// TIA Portal project "Polinka_3P_kwalifikacje_V16" (V16)

(* hardware
DEVICE "S7-1200 station_1"  S7-1200 Station
   slot 0: "Rack_0"  S7-1200 Rack  Rack  V1.0
   slot 1: "Polinka_Model"  CPU 1215C DC/DC/DC  6ES7 215-1AG40-0XB0  V4.2
DEVICE "S7-1200 station_2"  S7-1200 Station
   slot 0: "Rack_0"  S7-1200 Rack  Rack  V1.0
   slot 1: "Sterownik_do_zaprogramowania"  CPU 1215C DC/DC/DC  6ES7 215-1AG40-0XB0  V4.2
DEVICE "Polinka_HMI"  KTP700 Basic PN
   slot 0: "Polinka_HMI"  KTP700 Basic PN  6AV2 123-2GB03-0AX0  15.0.0.0
   slot 1: "HMI_RT_1"  KTP700 Basic PN  6AV2 123-2GB03-0AX0  15.0.0.0
   slot 5: "Polinka_HMI.IE_CP_1"  PROFINET Interface  15.0.0.0
      slot 1: "PROFINET Interface_1"  PROFINET Interface
         slot 1: "Port_1"  Port
*)

// ===== PLC "Polinka_Model"  CPU 1215C DC/DC/DC =====

VAR_GLOBAL   // PLC tag table "Default tag table"
   "System_Byte" AT %MB1 : Byte;
   "FirstScan" AT %M1.0 : Bool;
   "DiagStatusUpdate" AT %M1.1 : Bool;
   "AlwaysTRUE" AT %M1.2 : Bool;
   "AlwaysFALSE" AT %M1.3 : Bool;
   "Clock_Byte" AT %MB0 : Byte;
   "Clock_10Hz" AT %M0.0 : Bool;
   "Clock_5Hz" AT %M0.1 : Bool;
   "Clock_2.5Hz" AT %M0.2 : Bool;
   "Clock_2Hz" AT %M0.3 : Bool;
   "Clock_1.25Hz" AT %M0.4 : Bool;
   "Clock_1Hz" AT %M0.5 : Bool;
   "Clock_0.625Hz" AT %M0.6 : Bool;
   "Clock_0.5Hz" AT %M0.7 : Bool;
   "Tag_1" AT %M100.0 : Bool;
   "Tag_2" AT %M111.0 : Bool;
END_VAR

DATA_BLOCK "DB"   // DB1
{ S7_Optimized_Access := 'TRUE' }
VERSION : 0.1
   VAR
      w1_x : Int;
      w1_y : Int;
      w1_v : Real := 5.0;
      w1_drzwi_dx : Int := 0;
      w1_drzwiL_dx : Int;
      w1_drzwiP_dx : Int;
      w1_liczba_pasażerów : Int := 0;
      w1_drzwi_zamknięte : Bool;
      w1_drzwi_otwarte : Bool;
      zero : Int := 0;
      w2_y : Int := 0;
      w2_v : Int := 0;
      w2_drzwi_dx : Int := 0;
      w2_drzwiL_dx : Int := 0;
      w2_drzwiP_dx : Int := 0;
      w2_liczba_pasażerów : Int := 0;
      w2_drzwi_zamknięte : Bool := 0;
      w2_drzwi_otwarte : Bool := 0;
      w2_x : Int := 0;
      prędkość_wiatru : Real := 1.5;
      temperatura : Real := 20.0;
      czas_do_odjazdu : Int := 60;
      stacjaA_silnik_prędkość_zadana : Real := 0.0;
      stacjaA_silnik_prędkość_odczytana : Real := 0.0;
      stacjaA_silnik_przegrzanie : Bool;
      stacjaA_prędkość_odczytana : Real := 0.0;
      stacjaB_prędkość_odczytana : Real := 0.0;
      stacjaA_hamulec : Bool := false;
      stacjaB_hamulec : Bool := false;
      stacjaA_cz_A1 : Bool := false;
      stacjaA_cz_A2 : Bool := false;
      stacjaB_cz_B1 : Bool := false;
      stacjaB_cz_B2 : Bool := false;
      w1_d : Real := 0.0;
      w2_d : Real := 0.0;
      stacjaA_pasażer_0 : Bool := false;
      "stacjaA_pasażer+1" : Bool := false;
      "stacjaA_pasażer-1" : Bool := false;
      stacjaA_pasażerUP : Bool;
      stacjaA_pasażerDOWN : Bool;
      stacjaB_pasażer_0 : Bool := false;
      "stacjaB_pasażer+1" : Bool := false;
      "stacjaB_pasażer-1" : Bool := false;
      stacjaB_pasażerUP : Bool;
      stacjaB_pasażerDOWN : Bool;
      klawiatura : Word;
      awaria5 : Bool := false;
      awaria4 : Bool := false;
      awaria3 : Bool := false;
      awaria2 : Bool := false;
      awaria1 : Bool := false;
   END_VAR
BEGIN
END_DATA_BLOCK

DATA_BLOCK "Polinka_DB"   // DB2
{ S7_Optimized_Access := 'FALSE' }
VERSION : 0.1
   VAR
      st_stacjaA_silnik_prędkość : Real := 0.0;   // sterowanie prędkością silnika
      st_stacjaA_hamulec : Bool := true;   // sterowanie: 1 - hamulec włączony; 0 - wyłączony w stacji A
      st_stacjaA_zielone : Bool := false;   // sygnalizacja świetlna: 1-dozwolone wejście do wagonika
      st_stacjaA_czerwone : Bool := false;   // sygnalizacja świetlna: 1-zabronione wejście do wagonika
      st_stacjaB_hamulec : Bool := true;   // sterowanie: 1 - hamulec włączony; 0 - wyłączony w stacji B
      st_stacjaB_zielone : Bool := false;   // sygnalizacja świetlna: 1-dozwolone wejście do wagonika
      st_stacjaB_czerwone : Bool := false;   // sygnalizacja świetlna: 1-zabronione wejście do wagonika
      st_wagonik1_drzwi_zamykaj : Bool := false;   // 1 - zamykaj drzwi w wagoniku 1
      st_wagonik1_drzwi_otwieraj : Bool := false;   // 1 - otwieraj drzwi w wagoniku 1
      st_wagonik2_drzwi_zamykaj : Bool := false;   // 1 - zamykaj drzwi w wagoniku 2
      st_wagonik2_drzwi_otwieraj : Bool := false;   // 1 - otwieraj drzwi w wagoniku 2
      st_czas_do_odjazdu : Int := 60;   // czas pozostały do odjazdu wagoników
      st_kontrolka_STOP : Bool := false;   // 1 - podświetlaj przycisk "STOP"
      st_kontrolka_AUTO : Bool := false;   // 1 - podświetlaj przycisk "AUTO"
      st_kontrolka_RĘCZNIE : Bool := false;   // 1 - podświetlaj przycisk "RĘCZNIE"
      cz_wagonik1_położenie : Real;   // położenie wagonika 1, 0m - w stacji A, 756m - w stacji B
      "cz_wagonik1_l.pasażerów" : Int;   // liczba pasażerów w wagoniku 1
      cz_wagonik1_DZ : Bool;   // 1 gdy Drzwi w pełni Zamknięte i zabezpieczone
      cz_wagonik1_DO : Bool;   // 1 gdy Drzwi w pełni Otwarte i zabezpieczone
      cz_wagonik2_położenie : Real;   // położenie wagonika 2, 0m - w stacji A, 756m - w stacji B
      "cz_wagonik2_l.pasażerów" : Int;   // liczba pasażerów w wagoniku 2
      cz_wagonik2_DZ : Bool;   // 1 gdy Drzwi w pełni Zamknięte i zabezpieczone
      cz_wagonik2_DO : Bool;   // 1 gdy Drzwi w pełni Otwarte i zabezpieczone
      "cz_stacjaA_prędkość_(silnik)" : Real;   // prędkość liny napędowej odczytana na wale silnika [m/s]
      cz_stacjaA_prędkość : Real;   // prędkość liny napędowej odczytana w stacji A [m/s]
      cz_stacjaA_temperatura : Real;   // temperatura zewnętrzna
      cz_stacjaA_wiatr : Real;   // prędkość wiatru
      cz_stacjaA_silnik_przegrzanie : Bool;   // 1: działanie zabezpieczenia termicznego silnika
      cz_stacjaA_A1 : Bool;   // 1: wagonik na przystanku w stacji A
      cz_stacjaA_A2 : Bool;   // 1: wykolejona lina napędowa na słupie w stacji A
      cz_stacjaB_prędkość : Real;   // prędkość liny napędowej odczytana w stacji B [m/s]
      cz_stacjaB_B1 : Bool;   // 1: wagonik na przystanku w stacji B
      cz_stacjaB_B2 : Bool;   // 1: wykolejona lina napędowa na słupie w stacji B
      p_STOP : Bool;   // przycisk monostabilny STOP
      p_AUTO : Bool;   // przycisk monostabilny AUTO
      p_RĘCZNE : Bool;   // przycisk monostabilny RĘCZNIE
      "p_prędkość-20" : Bool;   // przycisk monostabilny -20 m/s
      "p_prędkość-5" : Bool;   // przycisk monostabilny -5 m/s
      p_prędkość_0 : Bool;   // przycisk monostabilny 0 m/s
      "p_prędkość+5" : Bool;   // przycisk monostabilny +5 m/s
      "p_prędkość+20" : Bool;   // przycisk monostabilny +20 m/s
      p_hamulecA_zał : Bool;   // przycisk monostabilny Hamulec A załącz
      p_hamulecA_wył : Bool;   // przycisk monostabilny Hamulec A wyłącz
      p_hamulecB_zał : Bool;   // przycisk monostabilny Hamulec B załącz
      p_hamulecB_wył : Bool;   // przycisk monostabilny Hamulec B wyłącz
      p_wagonik1_otw : Bool;   // przycisk mono.: otwieraj drzwi w wagoniku 1
      p_wagonik1_zam : Bool;   // przycisk mono.: zamykaj drzwi w wagoniku 1
      p_wagonik2_otw : Bool;   // przycisk mono.: otwieraj drzwi w wagoniku 2
      p_wagonik2_zam : Bool;   // przycisk mono.: zamykaj drzwi w wagoniku 2
   END_VAR
BEGIN
END_DATA_BLOCK

FUNCTION "fun3_Ruch_wagoników" : Void   // FC1, SCL
{ S7_Optimized_Access := 'TRUE' }
VERSION : 0.1
   VAR_TEMP
      d1 : Real;
      d2 : Real;
      d3 : Real;
      d4 : Real;
      d5 : Real;
      v_skala : Real;
      dk : Real;
      d : Real;
   END_VAR
   VAR CONSTANT
      "dT" : Real := 0.1;   // krok czasowy symulacji modelu [sek]
   END_VAR
BEGIN
   #v_skala := 1.0;

   #d1 := 20.0;
   #d2 := 158.0;
   #d3 := 400.0;
   #d4 := 158.0;
   #d5 := 20.0;

   #d := #d1 + #d2 + #d3 + #d4 + #d5 - (#d2 - 124.0) - (#d4 - 124.0);

   // 1. wagonik 1 - żółty:
   "DB".w1_d := "DB".w1_d + "DB".w1_v * #v_skala * #dT;
   IF "DB".w1_d < -18 THEN
       "DB".w1_d := -18;
   END_IF;

   IF "DB".w1_d > #d1 + #d2 + #d3 + #d4 + #d5 + 18.0 THEN
       "DB".w1_d := #d1 + #d2 + #d3 + #d4 + #d5 + 18.0;
   END_IF;

   // ruch na stacji A
   IF "DB".w1_d < #d1 THEN
       "DB".w1_x := "DB".w1_d;
       "DB".w1_y := 0.0;
   END_IF;

   // od stacji A do lewego słupa
   IF ("DB".w1_d >= #d1) AND ("DB".w1_d < #d1 + #d2)THEN
       #dk := "DB".w1_d - #d1;
       "DB".w1_y := -100.0 * #dk / #d2;
       "DB".w1_x := #d1 + 124.0 * #dk / #d2;
   END_IF;

   // między słupami
   IF ("DB".w1_d >= #d1 + #d2) AND ("DB".w1_d < #d1 + #d2 + #d3) THEN
       "DB".w1_x := "DB".w1_d - (#d2 - 124.0);
       "DB".w1_y := -100.0;
   END_IF;

   // od prawego słupa do stacji B
   IF ("DB".w1_d >= #d1 + #d2 + #d3) AND ("DB".w1_d < #d1 + #d2 + #d3 + #d4) THEN
       #dk := "DB".w1_d - #d1 - #d2 - #d3;
       "DB".w1_y := -100.0 + 100.0 * #dk / #d4;

       "DB".w1_x := "DB".w1_d - (#d2 - 124.0) + 124.0 * #dk / #d4;
       "DB".w1_x := #d1 + (#d2 - 34.0) + #d3 + 124.0 * #dk / #d4;
   END_IF;

   // ruch na stacji B
   IF ("DB".w1_d >= #d1 + #d2 + #d3 + #d4) THEN
       "DB".w1_x := "DB".w1_d - (#d2 - 124.0) - (#d4 - 124.0);
       "DB".w1_y := 0.0;
   END_IF;


   //  wagonik 2 - czerwony:
   "DB".w2_y := "DB".w1_y;
   "DB".w2_x := #d - "DB".w1_x;
   "DB".w2_x := -"DB".w1_x;
   "DB".w2_d := #d1 + #d2 + #d3 + #d4 + #d5 - "DB".w1_d;


   //krańcówki cz_A1 i cz_A2
   IF ("DB".w1_d <= 0) OR ("DB".w2_d <= 0) THEN
       "DB".stacjaA_cz_A1 := TRUE;
   ELSE
       "DB".stacjaA_cz_A1 := FALSE;
   END_IF;

   IF ("DB".w1_d >= 756) OR ("DB".w2_d >= 756) THEN
       "DB".stacjaB_cz_B1 := TRUE;
   ELSE
       "DB".stacjaB_cz_B1 := FALSE;
   END_IF;
END_FUNCTION

FUNCTION "fun4_Drzwi_wagoników" : Void   // FC2, SCL
{ S7_Optimized_Access := 'TRUE' }
VERSION : 0.1
BEGIN
   // wagonik 1 - drzwi:
   IF "Polinka_DB".st_wagonik1_drzwi_otwieraj THEN
       "DB".w1_drzwi_dx := "DB".w1_drzwi_dx + 1;
   END_IF;

   IF "Polinka_DB".st_wagonik1_drzwi_zamykaj THEN
       "DB".w1_drzwi_dx := "DB".w1_drzwi_dx - 1;
   END_IF;

   "DB".w1_drzwi_zamknięte := FALSE;
   "DB".w1_drzwi_otwarte := FALSE;
   IF "DB".w1_drzwi_dx <=0 THEN
       "DB".w1_drzwi_dx := 0;
       "DB".w1_drzwi_zamknięte := true;
   END_IF;

   IF "DB".w1_drzwi_dx >= 14 THEN
       "DB".w1_drzwi_dx := 14;
       "DB".w1_drzwi_otwarte := true;
   END_IF;

   "DB".w1_drzwiP_dx := "DB".w1_x + "DB".w1_drzwi_dx;
   "DB".w1_drzwiL_dx := "DB".w1_x - "DB".w1_drzwi_dx;

   // Błędne sterowanie (obie linie aktywne):
   IF "Polinka_DB".st_wagonik1_drzwi_zamykaj AND "Polinka_DB".st_wagonik1_drzwi_otwieraj THEN
       "DB".w1_drzwi_zamknięte := TRUE;
       "DB".w1_drzwi_otwarte := TRUE;
   END_IF;



   // wagonik 2 - drzwi:
   IF "Polinka_DB".st_wagonik2_drzwi_otwieraj THEN
       "DB".w2_drzwi_dx := "DB".w2_drzwi_dx + 1;
   END_IF;

   IF "Polinka_DB".st_wagonik2_drzwi_zamykaj THEN
       "DB".w2_drzwi_dx := "DB".w2_drzwi_dx - 1;
   END_IF;

   "DB".w2_drzwi_zamknięte := FALSE;
   "DB".w2_drzwi_otwarte := FALSE;
   IF "DB".w2_drzwi_dx <= 0 THEN
       "DB".w2_drzwi_dx := 0;
       "DB".w2_drzwi_zamknięte := true;
   END_IF;

   IF "DB".w2_drzwi_dx >= 14 THEN
       "DB".w2_drzwi_dx := 14;
       "DB".w2_drzwi_otwarte := true;
   END_IF;

   "DB".w2_drzwiP_dx := "DB".w2_x + "DB".w2_drzwi_dx;
   "DB".w2_drzwiL_dx := "DB".w2_x - "DB".w2_drzwi_dx;

   // Błędne sterowanie (obie linie aktywne):
   IF "Polinka_DB".st_wagonik2_drzwi_zamykaj AND "Polinka_DB".st_wagonik2_drzwi_otwieraj THEN
       "DB".w2_drzwi_zamknięte := TRUE;
       "DB".w2_drzwi_otwarte := TRUE;
   END_IF;



   ///
   (*
   // wagonik 1 - drzwi:
   IF "Polinka_DB".st_wagonik1_drzwi_otwieraj THEN
       "DB".w1_drzwi_dx := "DB".w1_drzwi_dx + 1;
   END_IF;

   IF "Polinka_DB".st_wagonik1_drzwi_zamykaj THEN
       "DB".w1_drzwi_dx := "DB".w1_drzwi_dx - 1;
   END_IF;

   "Polinka_DB".cz_wagonik1_DZ := FALSE;
   "Polinka_DB".cz_wagonik1_DO := FALSE;
   IF "DB".w1_drzwi_dx <=0 THEN
       "DB".w1_drzwi_dx := 0;
       "Polinka_DB".cz_wagonik1_DZ := true;
   END_IF;

   IF "DB".w1_drzwi_dx >= 14 THEN
       "DB".w1_drzwi_dx := 14;
       "Polinka_DB".cz_wagonik1_DO := true;
   END_IF;

   "DB".w1_drzwiP_dx := "DB".w1_x + "DB".w1_drzwi_dx;
   "DB".w1_drzwiL_dx := "DB".w1_x - "DB".w1_drzwi_dx;

   // Błędne sterowanie (obie linie aktywne):
   IF "Polinka_DB".st_wagonik1_drzwi_zamykaj AND "Polinka_DB".st_wagonik1_drzwi_otwieraj THEN
       "Polinka_DB".cz_wagonik1_DZ := TRUE;
       "Polinka_DB".cz_wagonik1_DO := TRUE;
   END_IF;



   // wagonik 2 - drzwi:
   IF "Polinka_DB".st_wagonik2_drzwi_otwieraj THEN
       "DB".w2_drzwi_dx := "DB".w2_drzwi_dx + 1;
   END_IF;

   IF "Polinka_DB".st_wagonik2_drzwi_zamykaj THEN
       "DB".w2_drzwi_dx := "DB".w2_drzwi_dx - 1;
   END_IF;

   "Polinka_DB".cz_wagonik2_DZ := FALSE;
   "Polinka_DB".cz_wagonik2_DO := FALSE;
   IF "DB".w2_drzwi_dx <= 0 THEN
       "DB".w2_drzwi_dx := 0;
       "Polinka_DB".cz_wagonik2_DZ := true;
   END_IF;

   IF "DB".w2_drzwi_dx >= 14 THEN
       "DB".w2_drzwi_dx := 14;
       "Polinka_DB".cz_wagonik2_DO := true;
   END_IF;

   "DB".w2_drzwiP_dx := "DB".w2_x + "DB".w2_drzwi_dx;
   "DB".w2_drzwiL_dx := "DB".w2_x - "DB".w2_drzwi_dx;

   // Błędne sterowanie (obie linie aktywne):
   IF "Polinka_DB".st_wagonik2_drzwi_zamykaj AND "Polinka_DB".st_wagonik2_drzwi_otwieraj THEN
       "Polinka_DB".cz_wagonik2_DZ := TRUE;
       "Polinka_DB".cz_wagonik2_DO := TRUE;
   END_IF;
   *)
END_FUNCTION

FUNCTION "fun5_Pasażerowie" : Void   // FC3, SCL
{ S7_Optimized_Access := 'TRUE' }
VERSION : 0.1
BEGIN
   "DB".stacjaA_pasażerDOWN := FALSE;
   "DB".stacjaA_pasażerUP :=FALSE;
   "DB".stacjaB_pasażerDOWN := FALSE;
   "DB".stacjaB_pasażerUP := FALSE;

   (*
   IF "DB"."stacjaB_pasażer+1" OR "DB"."stacjaB_pasażer-1" OR "DB".stacjaB_pasażer_0 THEN
       "DB".czas_do_odjazdu := "DB".czas_do_odjazdu + 1;
   END_IF;
   *)


   // 1. wagonik 1 na stacji A:
   IF "DB".w1_d <= 0 (*AND "DB".w1_d >=-5*) THEN
       IF "Polinka_DB".cz_wagonik1_DO THEN

           "DB".stacjaA_pasażerDOWN := true;

           IF "DB"."stacjaA_pasażer-1" THEN
               "DB"."stacjaA_pasażer-1" := 0;
               "DB".w1_liczba_pasażerów := "DB".w1_liczba_pasażerów - 1;
               IF "DB".w1_liczba_pasażerów < 0 THEN
                   "DB".w1_liczba_pasażerów := 0;
               END_IF;
           END_IF;

           IF "DB"."stacjaA_pasażer_0" THEN
               "DB"."stacjaA_pasażer_0" := 0;
               "DB".w1_liczba_pasażerów := 0;
           END_IF;


           IF "Polinka_DB".st_stacjaA_zielone AND NOT  "Polinka_DB".st_stacjaA_czerwone THEN
               "DB".stacjaA_pasażerUP := true;
               IF "DB"."stacjaA_pasażer+1" THEN
                   "DB"."stacjaA_pasażer+1" := 0;
                   "DB".w1_liczba_pasażerów := "DB".w1_liczba_pasażerów + 1;
               END_IF;
           END_IF;

       END_IF;
   END_IF;


   // 2. wagonik 1 na stacji B:
   IF (*"DB".w1_d <= 762 AND*) "DB".w1_d >= 756 THEN
       IF "Polinka_DB".cz_wagonik1_DO THEN

           "DB".stacjaB_pasażerDOWN := true;

           IF "DB"."stacjaB_pasażer-1" THEN
               "DB"."stacjaB_pasażer-1" := 0;
               "DB".w1_liczba_pasażerów := "DB".w1_liczba_pasażerów - 1;
               IF "DB".w1_liczba_pasażerów < 0 THEN
                   "DB".w1_liczba_pasażerów := 0;
               END_IF;
           END_IF;

           IF "DB"."stacjaB_pasażer_0" THEN
               "DB"."stacjaB_pasażer_0" := 0;
               "DB".w1_liczba_pasażerów := 0;
           END_IF;


           IF "Polinka_DB".st_stacjaB_zielone AND NOT "Polinka_DB".st_stacjaB_czerwone THEN
               "DB".stacjaB_pasażerUP := true;
               IF "DB"."stacjaB_pasażer+1" THEN
                   "DB"."stacjaB_pasażer+1" := 0;
                   "DB".w1_liczba_pasażerów := "DB".w1_liczba_pasażerów + 1;
               END_IF;
           END_IF;

       END_IF;
   END_IF;


   // 3. wagonik 2 na stacji A:
   IF "DB".w2_d <= 0 (*AND "DB".w2_d >= -5*) THEN
       IF "Polinka_DB".cz_wagonik2_DO THEN

           "DB".stacjaA_pasażerDOWN := true;

           IF "DB"."stacjaA_pasażer-1" THEN
               "DB"."stacjaA_pasażer-1" := 0;
               "DB".w2_liczba_pasażerów := "DB".w2_liczba_pasażerów - 1;
               IF "DB".w2_liczba_pasażerów < 0 THEN
                   "DB".w2_liczba_pasażerów := 0;
               END_IF;
           END_IF;

           IF "DB"."stacjaA_pasażer_0" THEN
               "DB"."stacjaA_pasażer_0" := 0;
               "DB".w2_liczba_pasażerów := 0;
           END_IF;


           IF "Polinka_DB".st_stacjaA_zielone AND NOT "Polinka_DB".st_stacjaA_czerwone THEN
               "DB".stacjaA_pasażerUP := true;
               IF "DB"."stacjaA_pasażer+1" THEN
                   "DB"."stacjaA_pasażer+1" := 0;
                   "DB".w2_liczba_pasażerów := "DB".w2_liczba_pasażerów + 1;
               END_IF;
           END_IF;

       END_IF;
   END_IF;


   // 4. wagonik 2 na stacji B:
   IF (*"DB".w2_d <= 762 AND*) "DB".w2_d >= 756 THEN
       IF "Polinka_DB".cz_wagonik2_DO THEN

           "DB".stacjaB_pasażerDOWN := true;

           IF "DB"."stacjaB_pasażer-1" THEN
               "DB"."stacjaB_pasażer-1" := 0;
               "DB".w2_liczba_pasażerów := "DB".w2_liczba_pasażerów - 1;
               IF "DB".w2_liczba_pasażerów < 0 THEN
                   "DB".w2_liczba_pasażerów := 0;
               END_IF;
           END_IF;

           IF "DB"."stacjaB_pasażer_0" THEN
               "DB"."stacjaB_pasażer_0" := 0;
               "DB".w2_liczba_pasażerów := 0;
           END_IF;


           IF "Polinka_DB".st_stacjaB_zielone AND NOT "Polinka_DB".st_stacjaB_czerwone THEN
               "DB".stacjaB_pasażerUP := true;
               IF "DB"."stacjaB_pasażer+1" THEN
                   "DB"."stacjaB_pasażer+1" := 0;
                   "DB".w2_liczba_pasażerów := "DB".w2_liczba_pasażerów + 1;
               END_IF;
           END_IF;

       END_IF;
   END_IF;



   (*        
   "DB"."stacjaA_pasażer+1" := 0;
   "DB"."stacjaA_pasażer-1" := 0;
   "DB"."stacjaA_pasażer_0" := 0;
   "DB"."stacjaB_pasażer+1" := 0;
   "DB"."stacjaB_pasażer-1" := 0;
   "DB"."stacjaB_pasażer_0" := 0;
   *)
END_FUNCTION

FUNCTION "fun6_SynchronizujDB_OUT" : Void   // FC4, SCL
{ S7_Optimized_Access := 'TRUE' }
VERSION : 0.1
   VAR_TEMP
      "a" : Word;
   END_VAR
BEGIN
   (*
   //1. synchronizacja z PLC_2 do modelu
   // 1.1 prędkości
   "DB".stacjaA_silnik_prędkość_zadana := "Polinka_DB".st_stacjaA_silnik_prędkość;
   "DB".stacjaA_silnik_prędkość_odczytana := "Polinka_DB".st_stacjaA_silnik_prędkość;
   "DB".stacjaA_prędkość_odczytana := "Polinka_DB".st_stacjaA_silnik_prędkość;
   "DB".stacjaB_prędkość_odczytana := "Polinka_DB".st_stacjaA_silnik_prędkość;

   // 1.2 hamulce
   "DB".stacjaA_hamulec := "Polinka_DB".st_stacjaA_hamulec;
   "DB".stacjaB_hamulec := "Polinka_DB".st_stacjaB_hamulec;

   // inne
   "DB".czas_do_odjazdu := "Polinka_DB".st_czas_do_odjazdu;
   *)


   /////////////////////////////////////////////////////////////////////////////////////
   //2. synchronizacja z modelu do PLC_2
   // 2.1 prędkości
   "Polinka_DB"."cz_stacjaA_prędkość_(silnik)" := "DB".stacjaA_silnik_prędkość_odczytana;
   "Polinka_DB"."cz_stacjaA_prędkość" := "DB".stacjaA_prędkość_odczytana;
   "Polinka_DB"."cz_stacjaB_prędkość" := "DB".stacjaB_prędkość_odczytana;


   // 2.2 informacje o wagonikach
   "Polinka_DB".cz_wagonik1_położenie := "DB".w1_d;
   "Polinka_DB".cz_wagonik2_położenie := "DB".w2_d;

   "Polinka_DB"."cz_wagonik1_l.pasażerów" := "DB".w1_liczba_pasażerów;
   "Polinka_DB"."cz_wagonik2_l.pasażerów" := "DB".w2_liczba_pasażerów;

   "Polinka_DB"."cz_wagonik1_DZ" := "DB".w1_drzwi_zamknięte;
   "Polinka_DB"."cz_wagonik1_DO" := "DB".w1_drzwi_otwarte;
   "Polinka_DB"."cz_wagonik2_DZ" := "DB".w2_drzwi_zamknięte;
   "Polinka_DB"."cz_wagonik2_DO" := "DB".w2_drzwi_otwarte;


   // 2.3 klawatura Panelu sterującego (do sterowania ręcznego)
   IF ("DB".klawiatura AND 1) > 0 THEN
       "Polinka_DB".p_STOP := 1;
   ELSE
       "Polinka_DB".p_STOP := 0;
   END_IF;

   IF ("DB".klawiatura AND 2) > 0 THEN
       "Polinka_DB".p_AUTO := 1;
   ELSE
       "Polinka_DB".p_AUTO := 0;
   END_IF;

   IF ("DB".klawiatura AND 4) > 0 THEN
       "Polinka_DB".p_RĘCZNE := 1;
   ELSE
       "Polinka_DB".p_RĘCZNE := 0;
   END_IF;

   IF ("DB".klawiatura AND 8) > 0 THEN
       "Polinka_DB"."p_prędkość-20" := 1;
   ELSE
       "Polinka_DB"."p_prędkość-20" := 0;
   END_IF;

   IF ("DB".klawiatura AND 16) > 0 THEN
       "Polinka_DB"."p_prędkość-5" := 1;
   ELSE
       "Polinka_DB"."p_prędkość-5" := 0;
   END_IF;

   IF ("DB".klawiatura AND 32) > 0 THEN
       "Polinka_DB"."p_prędkość_0" := 1;
   ELSE
       "Polinka_DB"."p_prędkość_0" := 0;
   END_IF;

   IF ("DB".klawiatura AND 64) > 0 THEN
       "Polinka_DB"."p_prędkość+5" := 1;
   ELSE
       "Polinka_DB"."p_prędkość+5" := 0;
   END_IF;

   IF ("DB".klawiatura AND 128) > 0 THEN
       "Polinka_DB"."p_prędkość+20" := 1;
   ELSE
       "Polinka_DB"."p_prędkość+20" := 0;
   END_IF;

   IF ("DB".klawiatura AND 256) > 0 THEN
       "Polinka_DB".p_hamulecA_zał := 1;
   ELSE
       "Polinka_DB".p_hamulecA_zał := 0;
   END_IF;

   IF ("DB".klawiatura AND 512) > 0 THEN
       "Polinka_DB".p_hamulecA_wył := 1;
   ELSE
       "Polinka_DB".p_hamulecA_wył := 0;
   END_IF;

   IF ("DB".klawiatura AND 1024) > 0 THEN
       "Polinka_DB".p_hamulecB_zał := 1;
   ELSE
       "Polinka_DB".p_hamulecB_zał := 0;
   END_IF;

   IF ("DB".klawiatura AND 2048) > 0 THEN
       "Polinka_DB".p_hamulecB_wył := 1;
   ELSE
       "Polinka_DB".p_hamulecB_wył := 0;
   END_IF;

   IF ("DB".klawiatura AND 4096) > 0 THEN
       "Polinka_DB".p_wagonik1_otw := 1;
   ELSE
       "Polinka_DB".p_wagonik1_otw := 0;
   END_IF;

   IF ("DB".klawiatura AND 8192) > 0 THEN
       "Polinka_DB".p_wagonik1_zam := 1;
   ELSE
       "Polinka_DB".p_wagonik1_zam := 0;
   END_IF;

   IF ("DB".klawiatura AND 16384) > 0 THEN
       "Polinka_DB".p_wagonik2_otw := 1;
   ELSE
       "Polinka_DB".p_wagonik2_otw := 0;
   END_IF;

   IF ("DB".klawiatura AND 32768) > 0 THEN
       "Polinka_DB".p_wagonik2_zam := 1;
   ELSE
       "Polinka_DB".p_wagonik2_zam := 0;
   END_IF;




   // 2.4 inne
   "Polinka_DB".cz_stacjaA_temperatura := "DB".temperatura ;
   IF "DB".prędkość_wiatru < 0 THEN
       "DB".prędkość_wiatru := 0.0;
   END_IF;
   "Polinka_DB".cz_stacjaA_wiatr := "DB".prędkość_wiatru;
   "Polinka_DB".cz_stacjaA_silnik_przegrzanie := "DB".stacjaA_silnik_przegrzanie;

   "Polinka_DB".cz_stacjaA_A1 := "DB".stacjaA_cz_A1;
   "Polinka_DB".cz_stacjaA_A2 := "DB".stacjaA_cz_A2;
   "Polinka_DB".cz_stacjaB_B1 := "DB".stacjaB_cz_B1;
   "Polinka_DB".cz_stacjaB_B2 := "DB".stacjaB_cz_B2;
END_FUNCTION

FUNCTION "fun1_SynchronizujDB_IN" : Void   // FC5, SCL
{ S7_Optimized_Access := 'TRUE' }
VERSION : 0.1
BEGIN
   /////////////////////////////////////////////////////////////////////////////////////
   //1. synchronizacja DB z PLC_2 do modelu
   // 1.1 prędkości
   "DB".stacjaA_silnik_prędkość_zadana := "Polinka_DB".st_stacjaA_silnik_prędkość;
   "DB".stacjaA_silnik_prędkość_odczytana := "Polinka_DB".st_stacjaA_silnik_prędkość;
   "DB".stacjaA_prędkość_odczytana := "Polinka_DB".st_stacjaA_silnik_prędkość;
   "DB".stacjaB_prędkość_odczytana := "Polinka_DB".st_stacjaA_silnik_prędkość;
   "DB".w1_v := "DB".stacjaA_silnik_prędkość_odczytana;

   // 1.2 hamulce
   "DB".stacjaA_hamulec := "Polinka_DB".st_stacjaA_hamulec;
   "DB".stacjaB_hamulec := "Polinka_DB".st_stacjaB_hamulec;

   // inne
   "DB".czas_do_odjazdu := "Polinka_DB".st_czas_do_odjazdu;
END_FUNCTION

FUNCTION "fun2_Awarie" : Void   // FC6, SCL
{ S7_Optimized_Access := 'TRUE' }
VERSION : 0.1
BEGIN
   // Awaria 1. - wykolejenie liny na słupie przy stacji A
   IF "DB".awaria1 THEN
       "DB".stacjaA_cz_A2 := TRUE;
   ELSE
       "DB".stacjaA_cz_A2 := FALSE;
   END_IF;


   // Awaria 2. - przegrzany silnik
   IF "DB".awaria2 THEN
       "DB".stacjaA_silnik_przegrzanie := TRUE;
   ELSE
       "DB".stacjaA_silnik_przegrzanie := FALSE;
   END_IF;


   // Awaria 3. - uszkodzona prądniczka tachometryczna w stacji B
   IF "DB".awaria3 THEN
       "DB".stacjaB_prędkość_odczytana := 0;
   END_IF;


   // Awaria 4. - uszkodzona sprzęgło przy silniku (połowa prędkości zadanej na kołach napędowych)
   IF "DB".awaria4 THEN
       "DB".stacjaA_prędkość_odczytana := "DB".stacjaA_silnik_prędkość_odczytana / 3;
       "DB".stacjaB_prędkość_odczytana := "DB".stacjaA_silnik_prędkość_odczytana / 3;
       "DB".w1_v := "DB".stacjaA_silnik_prędkość_odczytana / 3;
   END_IF;


   // Awaria 5. - (brak)
END_FUNCTION

ORGANIZATION_BLOCK "Main"   // OB1, LAD, ProgramCycle
TITLE = "Main Program Sweep (Cycle)"
{ S7_Optimized_Access := 'TRUE' }
VERSION : 0.1
   VAR_INPUT
      Initial_Call : Bool;   // Initial call of this OB
      Remanence : Bool;   // =True, if remanent data are available
   END_VAR
BEGIN
END_ORGANIZATION_BLOCK

ORGANIZATION_BLOCK "Polinka_model_Cyclic"   // OB30, SCL, CyclicInterrupt
{ S7_Optimized_Access := 'TRUE' }
VERSION : 0.1
   VAR_INPUT
      Initial_Call : Bool;   // Initial call of this OB
      Event_Count : Int;   // Events discarded
   END_VAR
BEGIN

   "fun1_SynchronizujDB_IN"();

   "fun2_Awarie"();

   "fun3_Ruch_wagoników"();

   "fun4_Drzwi_wagoników"();

   "fun5_Pasażerowie"();

   "fun6_SynchronizujDB_OUT"();
END_ORGANIZATION_BLOCK

// ===== PLC "Sterownik_do_zaprogramowania"  CPU 1215C DC/DC/DC =====

VAR_GLOBAL   // PLC tag table "Default tag table"
   "Tag_1" AT %M1.0 : Bool;
   "Clock_Byte" AT %MB0 : Byte;
   "Clock_10Hz" AT %M0.0 : Bool;
   "Clock_5Hz" AT %M0.1 : Bool;
   "Clock_2.5Hz" AT %M0.2 : Bool;
   "Clock_2Hz" AT %M0.3 : Bool;
   "Clock_1.25Hz" AT %M0.4 : Bool;
   "Clock_1Hz" AT %M0.5 : Bool;
   "Clock_0.625Hz" AT %M0.6 : Bool;
   "Clock_0.5Hz" AT %M0.7 : Bool;
   "Mem_Clock_1Hz" AT %M1.5 : Bool;
   "get_done" AT %M10.0 : Bool;
   "send" AT %M10.1 : Bool;
   "put_done" AT %M10.2 : Bool;
   "mem_get_done" AT %M10.3 : Bool;
   "mem_put_done" AT %M10.4 : Bool;
END_VAR

DATA_BLOCK "Polinka_DB"   // DB2
{ S7_Optimized_Access := 'FALSE' }
VERSION : 0.1
   VAR
      st_stacjaA_silnik_prędkość : Real := 0.0;   // sterowanie prędkością silnika
      st_stacjaA_hamulec : Bool := true;   // sterowanie: 1 - hamulec włączony; 0 - wyłączony w stacji A
      st_stacjaA_zielone : Bool := false;   // sygnalizacja świetlna: 1-dozwolone wejście do wagonika
      st_stacjaA_czerwone : Bool := false;   // sygnalizacja świetlna: 1-zabronione wejście do wagonika
      st_stacjaB_hamulec : Bool := true;   // sterowanie: 1 - hamulec włączony; 0 - wyłączony w stacji B
      st_stacjaB_zielone : Bool := false;   // sygnalizacja świetlna: 1-dozwolone wejście do wagonika
      st_stacjaB_czerwone : Bool := false;   // sygnalizacja świetlna: 1-zabronione wejście do wagonika
      st_wagonik1_drzwi_zamykaj : Bool := false;   // 1 - zamykaj drzwi w wagoniku 1
      st_wagonik1_drzwi_otwieraj : Bool := false;   // 1 - otwieraj drzwi w wagoniku 1
      st_wagonik2_drzwi_zamykaj : Bool := false;   // 1 - zamykaj drzwi w wagoniku 2
      st_wagonik2_drzwi_otwieraj : Bool := false;   // 1 - otwieraj drzwi w wagoniku 2
      st_czas_do_odjazdu : Int := 60;   // czas pozostały do odjazdu wagoników
      st_kontrolka_STOP : Bool := false;   // 1 - podświetlaj przycisk "STOP"
      st_kontrolka_AUTO : Bool := true;   // 1 - podświetlaj przycisk "AUTO"
      st_kontrolka_RĘCZNIE : Bool := false;   // 1 - podświetlaj przycisk "RĘCZNIE"
      cz_wagonik1_położenie : Real;   // położenie wagonika 1, 0m - w stacji A, 756m - w stacji B
      "cz_wagonik1_l.pasażerów" : Int;   // liczba pasażerów w wagoniku 1
      cz_wagonik1_DZ : Bool;   // 1 gdy Drzwi w pełni Zamknięte i zabezpieczone
      cz_wagonik1_DO : Bool;   // 1 gdy Drzwi w pełni Otwarte i zabezpieczone
      cz_wagonik2_położenie : Real;   // położenie wagonika 2, 0m - w stacji A, 756m - w stacji B
      "cz_wagonik2_l.pasażerów" : Int;   // liczba pasażerów w wagoniku 2
      cz_wagonik2_DZ : Bool;   // 1 gdy Drzwi w pełni Zamknięte i zabezpieczone
      cz_wagonik2_DO : Bool;   // 1 gdy Drzwi w pełni Otwarte i zabezpieczone
      "cz_stacjaA_prędkość_(silnik)" : Real;   // prędkość liny napędowej odczytana na wale silnika [m/s]
      cz_stacjaA_prędkość : Real;   // prędkość liny napędowej odczytana w stacji A [m/s]
      cz_stacjaA_temperatura : Real;   // temperatura zewnętrzna
      cz_stacjaA_wiatr : Real;   // prędkość wiatru
      cz_stacjaA_silnik_przegrzanie : Bool;   // 1: działanie zabezpieczenia termicznego silnika
      cz_stacjaA_A1 : Bool;   // 1: wagonik na przystanku w stacji A
      cz_stacjaA_A2 : Bool;   // 1: wykolejona lina napędowa na słupie w stacji A
      cz_stacjaB_prędkość : Real;   // prędkość liny napędowej odczytana w stacji B [m/s]
      cz_stacjaB_B1 : Bool;   // 1: wagonik na przystanku w stacji B
      cz_stacjaB_B2 : Bool;   // 1: wykolejona lina napędowa na słupie w stacji B
      p_STOP : Bool;   // przycisk monostabilny STOP
      p_AUTO : Bool;   // przycisk monostabilny AUTO
      p_RĘCZNE : Bool;   // przycisk monostabilny RĘCZNIE
      "p_prędkość-20" : Bool;   // przycisk monostabilny -20 m/s
      "p_prędkość-5" : Bool;   // przycisk monostabilny -5 m/s
      p_prędkość_0 : Bool;   // przycisk monostabilny 0 m/s
      "p_prędkość+5" : Bool;   // przycisk monostabilny +5 m/s
      "p_prędkość+20" : Bool;   // przycisk monostabilny +20 m/s
      p_hamulecA_zał : Bool;   // przycisk monostabilny Hamulec A załącz
      p_hamulecA_wył : Bool;   // przycisk monostabilny Hamulec A wyłącz
      p_hamulecB_zał : Bool;   // przycisk monostabilny Hamulec B załącz
      p_hamulecB_wył : Bool;   // przycisk monostabilny Hamulec B wyłącz
      p_wagonik1_otw : Bool;   // przycisk mono.: otwieraj drzwi w wagoniku 1
      p_wagonik1_zam : Bool;   // przycisk mono.: zamykaj drzwi w wagoniku 1
      p_wagonik2_otw : Bool;   // przycisk mono.: otwieraj drzwi w wagoniku 2
      p_wagonik2_zam : Bool;   // przycisk mono.: zamykaj drzwi w wagoniku 2
   END_VAR
BEGIN
END_DATA_BLOCK

DATA_BLOCK "praca_automatyczna_DB"   // DB3
{ S7_Optimized_Access := 'TRUE' }
VERSION : 0.1
// stored: InstanceOfName praca_automatyczna
"praca_automatyczna"
BEGIN
END_DATA_BLOCK

DATA_BLOCK "zmienne_DB"   // DB5
{ S7_Optimized_Access := 'TRUE' }
VERSION : 0.1
   VAR
      kierunek_jazdy : SInt := 1;
      praca_auto : Bool := true;
      praca_reczna : Bool;
      STOP : Bool;
      "mem_p-5" : Bool;
      "mem_p-20" : Bool;
      "mem_p+5" : Bool;
      "mem_p+20" : Bool;
      unieruchomienie_wiatr : Bool;   // Jeżeli bit ma stan wysoki to kolejka zostaje unieruchomiona na jedenj ze stacji (monostabilny)
      predkosc_wagonika_mocny_wiatr : Real := 1.0;   // Prędkość wagonika, jeżeli mocno wieje. Ogranicznik 0.5
      unieruchomienie_temp : Bool;
      unieruchomienie : Bool;
      mem_p_STOP : Bool;
      mem_p_AUTO : Bool;
      uzyto_stop : Bool;
      AWARIA_1 : Bool;
      AWARIA_2 : Bool;
      AWARIA_3 : Bool;
      AWARIA_4 : Bool;
      blokada_AUTO : Bool;
      praca_reczna_ograniczona : Bool;
      do_stacji : Bool;
   END_VAR
BEGIN
END_DATA_BLOCK

DATA_BLOCK "obsluga_awarii_DB"   // DB6
{ S7_Optimized_Access := 'TRUE' }
VERSION : 0.1
// stored: InstanceOfName obsluga_awarii
"obsluga_awarii"
BEGIN
END_DATA_BLOCK

DATA_BLOCK "obsluga_awarii_polinka_DB"   // DB7
{ S7_Optimized_Access := 'TRUE' }
VERSION : 0.1
// stored: InstanceOfName obsluga_awarii_polinka
"obsluga_awarii_polinka"
BEGIN
END_DATA_BLOCK

FUNCTION_BLOCK "praca_automatyczna"   // FB1, LAD
{ S7_Optimized_Access := 'TRUE' }
VERSION : 0.1
   VAR
      czas_jazdy : Time;
      jazda : Bool;
      gotowi : Bool;
      IEC_Timer_0_Instance : TON_TIME;
      time_slow_down : Time;
      bylo_pelne : Bool;
   END_VAR
   VAR_TEMP   // added for the SCL form of the ladder/FBD networks
      _w1 : Bool;
   END_VAR
BEGIN

REGION Network 1
   // Odliczanie sekund, a gdy jedziemy mierzenie czasu
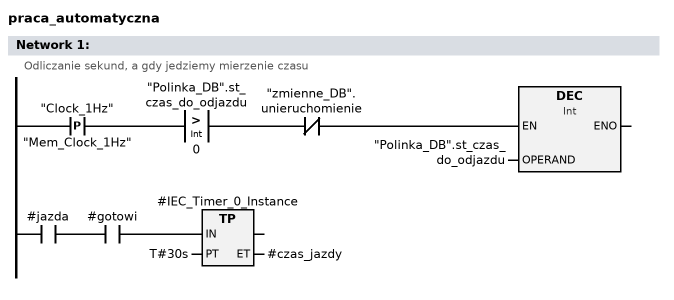
   #_w1 := "Clock_1Hz" AND NOT "Mem_Clock_1Hz";   // rising edge of "Clock_1Hz"
   "Mem_Clock_1Hz" := "Clock_1Hz";
   IF #_w1 AND ("Polinka_DB".st_czas_do_odjazdu > 0) AND NOT "zmienne_DB".unieruchomienie THEN
       "Polinka_DB".st_czas_do_odjazdu := "Polinka_DB".st_czas_do_odjazdu - 1;
   END_IF;
   #IEC_Timer_0_Instance(IN := #jazda AND #gotowi, PT := T#30s, ET => #czas_jazdy);   // TP
END_REGION

REGION Network 2 (SCL)
   // Jeśli skonczylo sie odliczanie, wagony nie są puste LUB jest 6 osób w obu wagonikach i nie #jazda to #jazda
   IF (("Polinka_DB".st_czas_do_odjazdu = 0 AND ("Polinka_DB"."cz_wagonik1_l.pasażerów" > 0 OR "Polinka_DB"."cz_wagonik2_l.pasażerów" > 0)) OR (("Polinka_DB"."cz_wagonik1_l.pasażerów" >= 6 AND "Polinka_DB"."cz_wagonik2_l.pasażerów" >= 6) AND NOT #bylo_pelne)) AND NOT #jazda AND NOT "zmienne_DB".unieruchomienie THEN
       #jazda := TRUE;
       "Polinka_DB".st_czas_do_odjazdu := 0;
       IF ("Polinka_DB"."cz_wagonik1_l.pasażerów" >= 6 AND "Polinka_DB"."cz_wagonik2_l.pasażerów" >= 6) THEN
           #bylo_pelne := TRUE;
       END_IF;
       // Zamknięcie drzwi w obu wagonikach
       "Polinka_DB".st_wagonik1_drzwi_otwieraj := 0;
       "Polinka_DB".st_wagonik2_drzwi_otwieraj := 0;
       "Polinka_DB".st_wagonik1_drzwi_zamykaj := 1;
       "Polinka_DB".st_wagonik2_drzwi_zamykaj := 1;
       // Zmiana światła na czerwone
       "Polinka_DB".st_stacjaA_zielone := 0;
       "Polinka_DB".st_stacjaA_czerwone := 1;
       "Polinka_DB".st_stacjaB_zielone := 0;
       "Polinka_DB".st_stacjaB_czerwone := 1;
       // Wyłączenie hamulcy
       "Polinka_DB".st_stacjaA_hamulec := 0;
       "Polinka_DB".st_stacjaB_hamulec := 0;
   // Gdy dalej trwa odliczanie:
   ELSIF NOT #jazda THEN
       // Drzwi otwarte w trakcie odliczania
       "Polinka_DB".st_wagonik1_drzwi_otwieraj := 1;
       "Polinka_DB".st_wagonik2_drzwi_otwieraj := 1;
       "Polinka_DB".st_wagonik1_drzwi_zamykaj := 0;
       "Polinka_DB".st_wagonik2_drzwi_zamykaj := 0;

       // Jeśli minął czas a nikogo nie ma to licz od początku
       IF "Polinka_DB".st_czas_do_odjazdu = 0 AND NOT ("Polinka_DB"."cz_wagonik1_l.pasażerów" > 0 OR "Polinka_DB"."cz_wagonik2_l.pasażerów" > 0) THEN
           "Polinka_DB".st_czas_do_odjazdu := 60;
       END_IF;
       // W zależności od kierunku jazdy wagoniki są na rożnych stacjach
       IF "zmienne_DB".kierunek_jazdy = 1 THEN
           // Jeśli pasażerów jest mniej niż 6 to zielone światło, w innym przypadku czerwone
           IF "Polinka_DB"."cz_wagonik1_l.pasażerów" < 6 THEN
               "Polinka_DB".st_stacjaA_zielone := 1;
               "Polinka_DB".st_stacjaA_czerwone := 0;
               #bylo_pelne := FALSE;
           ELSE
               "Polinka_DB".st_stacjaA_zielone := 0;
               "Polinka_DB".st_stacjaA_czerwone := 1;
           END_IF;
           IF "Polinka_DB"."cz_wagonik2_l.pasażerów" < 6 THEN
               "Polinka_DB".st_stacjaB_zielone := 1;
               "Polinka_DB".st_stacjaB_czerwone := 0;
               #bylo_pelne := FALSE;
           ELSE
               "Polinka_DB".st_stacjaB_zielone := 0;
               "Polinka_DB".st_stacjaB_czerwone := 1;
           END_IF;
       ELSE
           // Jeśli pasażerów jest mniej niż 6 to zielone światło, w innym przypadku czerwone
           IF "Polinka_DB"."cz_wagonik1_l.pasażerów" < 6 THEN
               "Polinka_DB".st_stacjaB_zielone := 1;
               "Polinka_DB".st_stacjaB_czerwone := 0;
               #bylo_pelne := FALSE;
           ELSE
               "Polinka_DB".st_stacjaB_zielone := 0;
               "Polinka_DB".st_stacjaB_czerwone := 1;
           END_IF;
           IF "Polinka_DB"."cz_wagonik2_l.pasażerów" < 6 THEN
               "Polinka_DB".st_stacjaA_zielone := 1;
               "Polinka_DB".st_stacjaA_czerwone := 0;
               #bylo_pelne := FALSE;
           ELSE
               "Polinka_DB".st_stacjaA_zielone := 0;
               "Polinka_DB".st_stacjaA_czerwone := 1;
           END_IF;
       END_IF;
   // Jeśli dojechał do końca to zatrzymaj, zmień kierunek oraz załącz hamulce
   ELSIF #jazda AND ("Polinka_DB".cz_stacjaA_A1 OR "Polinka_DB".cz_stacjaA_A2) AND #czas_jazdy > T#10s THEN
       #jazda := FALSE;
       "Polinka_DB".st_stacjaA_silnik_prędkość := 0;
       "zmienne_DB".kierunek_jazdy := - "zmienne_DB".kierunek_jazdy;
       "Polinka_DB".st_czas_do_odjazdu := 60;
       "Polinka_DB".st_czas_do_odjazdu := "Polinka_DB".st_czas_do_odjazdu + 1;
       // Załączenie hamulcy
       "Polinka_DB".st_stacjaA_hamulec := 1;
       "Polinka_DB".st_stacjaB_hamulec := 1;
   END_IF;
END_REGION

REGION Network 3 (SCL)
   // Gdy mamy jechać
   IF #jazda THEN
       // Najpierw sprawdzamy czy jesteśmy gotowi (zamknięte drzwi itp.)
       IF "Polinka_DB".cz_wagonik1_DZ AND "Polinka_DB".cz_wagonik2_DZ AND NOT "Polinka_DB".cz_wagonik1_DO
           AND NOT "Polinka_DB".cz_wagonik2_DO AND NOT "Polinka_DB".st_stacjaA_hamulec AND NOT "Polinka_DB".st_stacjaB_hamulec
           AND NOT "Polinka_DB".p_STOP THEN
           #gotowi := TRUE;
       ELSE
           #gotowi := FALSE;
       END_IF;
       // Gdy jesteśmy gotowi to w zależności od tego jak długo jedziemy tak zmieniamy prędkość
       IF #czas_jazdy < T#1s THEN
           #time_slow_down := T#0s;
           "Polinka_DB".st_stacjaA_silnik_prędkość := 0.0;
       ELSIF #czas_jazdy < T#2s THEN
           "Polinka_DB".st_stacjaA_silnik_prędkość := INT_TO_REAL("zmienne_DB".kierunek_jazdy) * 5.0;
       ELSIF #czas_jazdy < T#3s THEN
           "Polinka_DB".st_stacjaA_silnik_prędkość := INT_TO_REAL("zmienne_DB".kierunek_jazdy) * 25.0;
       ELSIF #czas_jazdy < T#4s THEN
           "Polinka_DB".st_stacjaA_silnik_prędkość := INT_TO_REAL("zmienne_DB".kierunek_jazdy) * 40.0;
       // Poniższy warunek oznacza tyle: wagonik jest dalej niż 70 m do celu
       ELSIF INT_TO_REAL("zmienne_DB".kierunek_jazdy) * "Polinka_DB".cz_wagonik1_położenie
           < INT_TO_REAL("zmienne_DB".kierunek_jazdy) * (378.0 + INT_TO_REAL("zmienne_DB".kierunek_jazdy) * 308.0) THEN
           "Polinka_DB".st_stacjaA_silnik_prędkość := INT_TO_REAL("zmienne_DB".kierunek_jazdy) * 50.0;
       // Odmierzamy czas od momentu gdy mamy zwalniać
       ELSIF #time_slow_down = T#0ms THEN
           #time_slow_down := #czas_jazdy;
       ELSIF #czas_jazdy < #time_slow_down + T#900ms THEN
           "Polinka_DB".st_stacjaA_silnik_prędkość := INT_TO_REAL("zmienne_DB".kierunek_jazdy) * 40.0;
       ELSIF #czas_jazdy < #time_slow_down + T#1900ms THEN
           "Polinka_DB".st_stacjaA_silnik_prędkość := INT_TO_REAL("zmienne_DB".kierunek_jazdy) * 25.0;
       ELSIF #czas_jazdy < #time_slow_down + T#2900ms THEN
           "Polinka_DB".st_stacjaA_silnik_prędkość := INT_TO_REAL("zmienne_DB".kierunek_jazdy) * 5.0;
       END_IF;
       "Polinka_DB".st_stacjaA_silnik_prędkość := "Polinka_DB".st_stacjaA_silnik_prędkość * "zmienne_DB".predkosc_wagonika_mocny_wiatr;
   END_IF;
END_REGION
END_FUNCTION_BLOCK

FUNCTION_BLOCK "Zadanie4"   // FB1, LAD
{ S7_Optimized_Access := 'TRUE' }
VERSION : 0.1
   VAR_INPUT
      cz_stacjaA_A2 : Bool;
      cz_stacjaA_silnik_przegrzanie : Bool;
      cz_stacjaA_prędkość : Real;
      cz_stacjaB_prędkość : Real;
      cz_stacjaA_A1 : Bool;
      cz_wagonik1_położenie : Real;
      pracaAuto : Bool;
      stacjaA_silnik_prędkość : Real;
      cz_stacjaA_prędkość_silnik : Real;
   END_VAR
   VAR_OUTPUT
      p_hamulecA_zal : Bool;
      p_hamulecA_Wyl : Bool;
      p_hamulecB_Wyl : Bool;
      p_hamulecB_zal : Bool;
      stopAwaryjny : Bool;
      blokadaPowrotuDoAuto : Bool;
      silnikPredkoscPrzeliczona : Real;
      reczneSterowanie : Bool;
   END_VAR
   VAR
      ALWAYS_ON : Bool := TRUE;
      setAwaria2 : Bool;
      setAwaria3 : Bool;
      manual1 : Bool;
      manual2 : Bool;
      resetAuto1 : Bool;
      resetAuto2 : Bool;
      speedADiv : Real;
      resetManual : Bool;
      speedBDiv : Real;
   END_VAR
   VAR_TEMP   // added for the SCL form of the ladder/FBD networks
      _w1 : Bool;
   END_VAR
BEGIN

REGION Network 1 (SCL): Przeliczenie wartości do porównania
   #speedADiv := #cz_stacjaA_prędkość_silnik / 3;
   #speedBDiv := #cz_stacjaA_prędkość_silnik / 3;
END_REGION

REGION Network 2: Załączenie blokady przejścia z trybu Manualnego do trybu automatyczneogo po Awarii
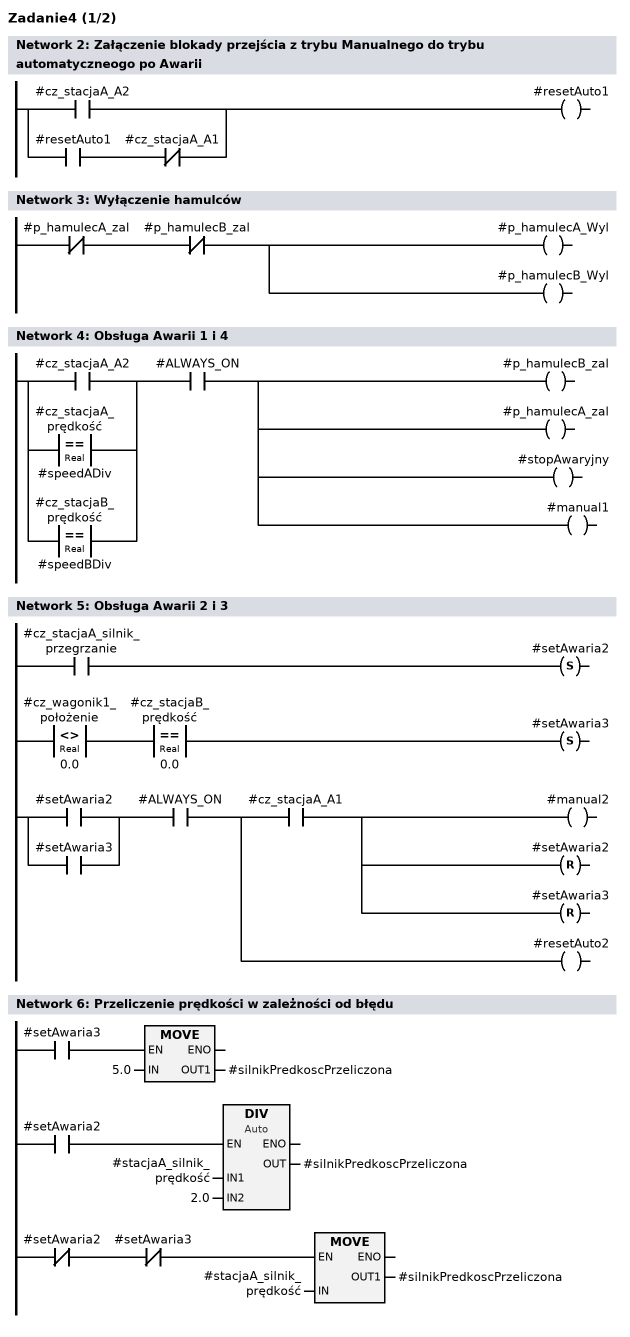
   RUNG wire#powerrail
      Contact( #cz_stacjaA_A2 )
      wire#w1
      Coil( #resetAuto1 )
   END_RUNG
   RUNG wire#powerrail
      Contact( #resetAuto1 )
      I_Contact( #cz_stacjaA_A1 )
   END_RUNG wire#w1
   // the same network as SCL:
   #resetAuto1 := #cz_stacjaA_A2 OR (#resetAuto1 AND NOT #cz_stacjaA_A1);
END_REGION

REGION Network 3: Wyłączenie hamulców
   RUNG wire#powerrail
      I_Contact( #p_hamulecA_zal )
      I_Contact( #p_hamulecB_zal )
      wire#w1
      Coil( #p_hamulecA_Wyl )
   END_RUNG
   RUNG wire#w1
      Coil( #p_hamulecB_Wyl )
   END_RUNG
   // the same network as SCL:
   #p_hamulecA_Wyl := NOT #p_hamulecA_zal AND NOT #p_hamulecB_zal;
   #p_hamulecB_Wyl := #p_hamulecA_Wyl;
END_REGION

REGION Network 4: Obsługa Awarii 1 i 4
   RUNG wire#powerrail
      Contact( #cz_stacjaA_A2 )
      wire#w1
      Contact( #ALWAYS_ON )
      wire#w2
      Coil( #p_hamulecB_zal )
   END_RUNG
   RUNG wire#powerrail
      { S7_Templates := "SrcType := Real" } EQ_Contact(in1 := #cz_stacjaA_prędkość, in2 := #speedADiv)
   END_RUNG wire#w1
   RUNG wire#powerrail
      { S7_Templates := "SrcType := Real" } EQ_Contact(in1 := #cz_stacjaB_prędkość, in2 := #speedBDiv)
   END_RUNG wire#w1
   RUNG wire#w2
      Coil( #p_hamulecA_zal )
   END_RUNG
   RUNG wire#w2
      Coil( #stopAwaryjny )
   END_RUNG
   RUNG wire#w2
      Coil( #manual1 )
   END_RUNG
   // the same network as SCL:
   #p_hamulecB_zal := (#cz_stacjaA_A2 OR (#cz_stacjaA_prędkość = #speedADiv) OR (#cz_stacjaB_prędkość = #speedBDiv)) AND #ALWAYS_ON;
   #p_hamulecA_zal := #p_hamulecB_zal;
   #stopAwaryjny := #p_hamulecB_zal;
   #manual1 := #p_hamulecB_zal;
END_REGION

REGION Network 5: Obsługa Awarii 2 i 3
   RUNG wire#powerrail
      Contact( #cz_stacjaA_silnik_przegrzanie )
      S_Coil( #setAwaria2 )
   END_RUNG
   RUNG wire#powerrail
      { S7_Templates := "SrcType := Real" } NE_Contact(in1 := #cz_wagonik1_położenie, in2 := 0.0)
      { S7_Templates := "SrcType := Real" } EQ_Contact(in1 := #cz_stacjaB_prędkość, in2 := 0.0)
      S_Coil( #setAwaria3 )
   END_RUNG
   RUNG wire#powerrail
      Contact( #setAwaria2 )
      wire#w1
      Contact( #ALWAYS_ON )
      wire#w2
      Contact( #cz_stacjaA_A1 )
      wire#w3
      Coil( #manual2 )
   END_RUNG
   RUNG wire#powerrail
      Contact( #setAwaria3 )
   END_RUNG wire#w1
   RUNG wire#w3
      R_Coil( #setAwaria2 )
   END_RUNG
   RUNG wire#w3
      R_Coil( #setAwaria3 )
   END_RUNG
   RUNG wire#w2
      Coil( #resetAuto2 )
   END_RUNG
   // the same network as SCL:
   IF #cz_stacjaA_silnik_przegrzanie THEN #setAwaria2 := TRUE; END_IF;
   IF (#cz_wagonik1_położenie <> 0.0) AND (#cz_stacjaB_prędkość = 0.0) THEN #setAwaria3 := TRUE; END_IF;
   #_w1 := (#setAwaria2 OR #setAwaria3) AND #ALWAYS_ON;
   #manual2 := #_w1 AND #cz_stacjaA_A1;
   IF #manual2 THEN
       #setAwaria2 := FALSE;
       #setAwaria3 := FALSE;
   END_IF;
   #resetAuto2 := #_w1;
END_REGION

REGION Network 6: Przeliczenie prędkości w zależności od błędu
   RUNG wire#powerrail
      Contact( #setAwaria3 )
      Move(in := 5.0, out1 => #silnikPredkoscPrzeliczona)
   END_RUNG
   RUNG wire#powerrail
      Contact( #setAwaria2 )
      Div(in1 := #stacjaA_silnik_prędkość, in2 := 2.0, out => #silnikPredkoscPrzeliczona)
   END_RUNG
   RUNG wire#powerrail
      I_Contact( #setAwaria2 )
      I_Contact( #setAwaria3 )
      Move(in := #stacjaA_silnik_prędkość, out1 => #silnikPredkoscPrzeliczona)
   END_RUNG
   // the same network as SCL:
   IF #setAwaria3 THEN #silnikPredkoscPrzeliczona := 5.0; END_IF;
   IF #setAwaria2 THEN #silnikPredkoscPrzeliczona := #stacjaA_silnik_prędkość / 2.0; END_IF;
   IF NOT #setAwaria2 AND NOT #setAwaria3 THEN
       #silnikPredkoscPrzeliczona := #stacjaA_silnik_prędkość;
   END_IF;
END_REGION

REGION Network 7: Zablokowanie przejścia z trybu Manualne do Automatycznego
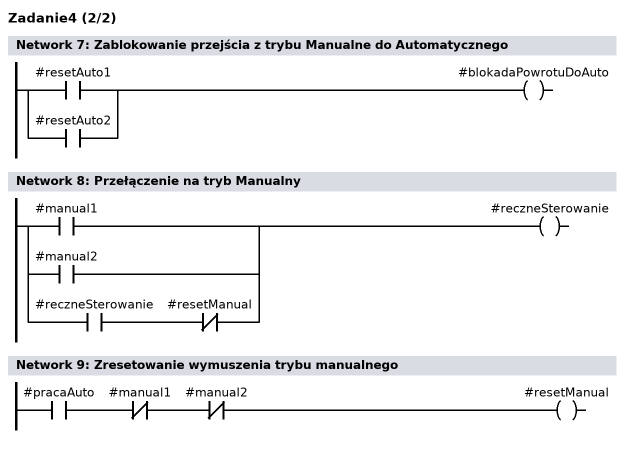
   RUNG wire#powerrail
      Contact( #resetAuto1 )
      wire#w1
      Coil( #blokadaPowrotuDoAuto )
   END_RUNG
   RUNG wire#powerrail
      Contact( #resetAuto2 )
   END_RUNG wire#w1
   // the same network as SCL:
   #blokadaPowrotuDoAuto := #resetAuto1 OR #resetAuto2;
END_REGION

REGION Network 8: Przełączenie na tryb Manualny
   RUNG wire#powerrail
      Contact( #manual1 )
      wire#w1
      Coil( #reczneSterowanie )
   END_RUNG
   RUNG wire#powerrail
      Contact( #manual2 )
   END_RUNG wire#w1
   RUNG wire#powerrail
      Contact( #reczneSterowanie )
      I_Contact( #resetManual )
   END_RUNG wire#w1
   // the same network as SCL:
   #reczneSterowanie := #manual1 OR #manual2 OR (#reczneSterowanie AND NOT #resetManual);
END_REGION

REGION Network 9: Zresetowanie wymuszenia trybu manualnego
   RUNG wire#powerrail
      Contact( #pracaAuto )
      I_Contact( #manual1 )
      I_Contact( #manual2 )
      Coil( #resetManual )
   END_RUNG
   // the same network as SCL:
   #resetManual := #pracaAuto AND NOT #manual1 AND NOT #manual2;
END_REGION
END_FUNCTION_BLOCK

FUNCTION_BLOCK "obsluga_awarii"   // FB2, LAD
{ S7_Optimized_Access := 'TRUE' }
VERSION : 0.1
   VAR_INPUT
      cz_stacjaA_A2 : Bool;
      cz_stacjaA_silnik_przegrzanie : Bool;
      cz_stacjaA_prędkość : Real;
      cz_stacjaB_prędkość : Real;
      cz_stacjaA_A1 : Bool;
      cz_wagonik1_położenie : Real;
      stacjaA_silnik_prędkość : Real;
      cz_stacjaA_prędkość_silnik : Real;
   END_VAR
   VAR_OUTPUT
      hamulecA_zal : Bool;
      hamulecB_zal : Bool;
      stopAwaryjny : Bool;
      blokadaPowrotuDoAuto : Bool;
      silnikPredkoscPrzeliczona : Real;
      reczneSterowanie : Bool;
      reczneOgraniczone : Bool;
   END_VAR
   VAR
      ALWAYS_ON : Bool := TRUE;
      setAwaria2 : Bool;
      setAwaria3 : Bool;
      manual1 : Bool;
      manual2 : Bool;
      resetAuto1 : Bool;
      resetAuto2 : Bool;
      speedADiv : Real;
      resetManual : Bool;
      speedBDiv : Real;
   END_VAR
BEGIN

REGION Network 1 (SCL): Przeliczenie wartości do porównania
   #speedADiv := #cz_stacjaA_prędkość_silnik / 3;
   #speedBDiv := #cz_stacjaA_prędkość_silnik / 3;
END_REGION

REGION Network 2: Załączenie blokady przejścia z trybu Manualnego do trybu automatyczneogo po Awarii
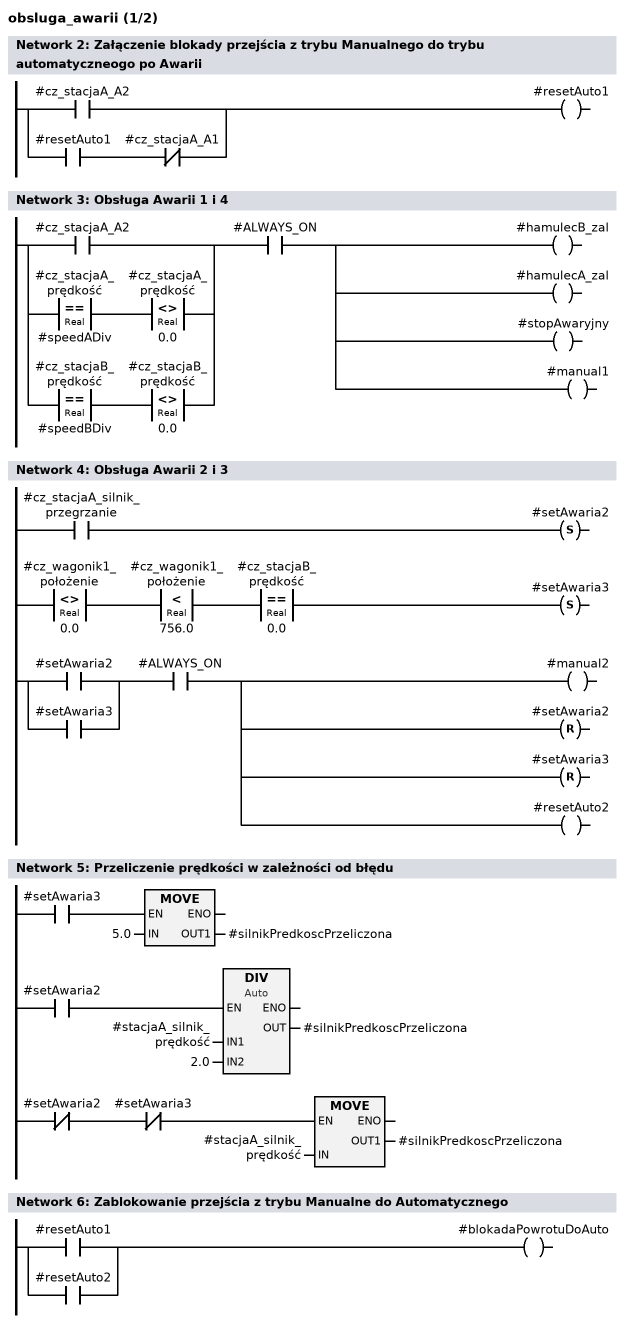
   RUNG wire#powerrail
      Contact( #cz_stacjaA_A2 )
      wire#w1
      Coil( #resetAuto1 )
   END_RUNG
   RUNG wire#powerrail
      Contact( #resetAuto1 )
      I_Contact( #cz_stacjaA_A1 )
   END_RUNG wire#w1
   // the same network as SCL:
   #resetAuto1 := #cz_stacjaA_A2 OR (#resetAuto1 AND NOT #cz_stacjaA_A1);
END_REGION

REGION Network 3: Obsługa Awarii 1 i 4
   RUNG wire#powerrail
      Contact( #cz_stacjaA_A2 )
      wire#w1
      Contact( #ALWAYS_ON )
      wire#w2
      Coil( #hamulecB_zal )
   END_RUNG
   RUNG wire#powerrail
      { S7_Templates := "SrcType := Real" } EQ_Contact(in1 := #cz_stacjaA_prędkość, in2 := #speedADiv)
      { S7_Templates := "SrcType := Real" } NE_Contact(in1 := #cz_stacjaA_prędkość, in2 := 0.0)
   END_RUNG wire#w1
   RUNG wire#powerrail
      { S7_Templates := "SrcType := Real" } EQ_Contact(in1 := #cz_stacjaB_prędkość, in2 := #speedBDiv)
      { S7_Templates := "SrcType := Real" } NE_Contact(in1 := #cz_stacjaB_prędkość, in2 := 0.0)
   END_RUNG wire#w1
   RUNG wire#w2
      Coil( #hamulecA_zal )
   END_RUNG
   RUNG wire#w2
      Coil( #stopAwaryjny )
   END_RUNG
   RUNG wire#w2
      Coil( #manual1 )
   END_RUNG
   // the same network as SCL:
   #hamulecB_zal := (#cz_stacjaA_A2 OR ((#cz_stacjaA_prędkość = #speedADiv) AND (#cz_stacjaA_prędkość <> 0.0)) OR ((#cz_stacjaB_prędkość = #speedBDiv) AND (#cz_stacjaB_prędkość <> 0.0))) AND #ALWAYS_ON;
   #hamulecA_zal := #hamulecB_zal;
   #stopAwaryjny := #hamulecB_zal;
   #manual1 := #hamulecB_zal;
END_REGION

REGION Network 4: Obsługa Awarii 2 i 3
   RUNG wire#powerrail
      Contact( #cz_stacjaA_silnik_przegrzanie )
      S_Coil( #setAwaria2 )
   END_RUNG
   RUNG wire#powerrail
      { S7_Templates := "SrcType := Real" } NE_Contact(in1 := #cz_wagonik1_położenie, in2 := 0.0)
      { S7_Templates := "SrcType := Real" } LT_Contact(in1 := #cz_wagonik1_położenie, in2 := 756.0)
      { S7_Templates := "SrcType := Real" } EQ_Contact(in1 := #cz_stacjaB_prędkość, in2 := 0.0)
      S_Coil( #setAwaria3 )
   END_RUNG
   RUNG wire#powerrail
      Contact( #setAwaria2 )
      wire#w1
      Contact( #ALWAYS_ON )
      wire#w2
      Coil( #manual2 )
   END_RUNG
   RUNG wire#powerrail
      Contact( #setAwaria3 )
   END_RUNG wire#w1
   RUNG wire#w2
      R_Coil( #setAwaria2 )
   END_RUNG
   RUNG wire#w2
      R_Coil( #setAwaria3 )
   END_RUNG
   RUNG wire#w2
      Coil( #resetAuto2 )
   END_RUNG
   // the same network as SCL:
   IF #cz_stacjaA_silnik_przegrzanie THEN #setAwaria2 := TRUE; END_IF;
   IF (#cz_wagonik1_położenie <> 0.0) AND (#cz_wagonik1_położenie < 756.0) AND (#cz_stacjaB_prędkość = 0.0) THEN
       #setAwaria3 := TRUE;
   END_IF;
   #manual2 := (#setAwaria2 OR #setAwaria3) AND #ALWAYS_ON;
   IF #manual2 THEN
       #setAwaria2 := FALSE;
       #setAwaria3 := FALSE;
   END_IF;
   #resetAuto2 := #manual2;
END_REGION

REGION Network 5: Przeliczenie prędkości w zależności od błędu
   RUNG wire#powerrail
      Contact( #setAwaria3 )
      Move(in := 5.0, out1 => #silnikPredkoscPrzeliczona)
   END_RUNG
   RUNG wire#powerrail
      Contact( #setAwaria2 )
      Div(in1 := #stacjaA_silnik_prędkość, in2 := 2.0, out => #silnikPredkoscPrzeliczona)
   END_RUNG
   RUNG wire#powerrail
      I_Contact( #setAwaria2 )
      I_Contact( #setAwaria3 )
      Move(in := #stacjaA_silnik_prędkość, out1 => #silnikPredkoscPrzeliczona)
   END_RUNG
   // the same network as SCL:
   IF #setAwaria3 THEN #silnikPredkoscPrzeliczona := 5.0; END_IF;
   IF #setAwaria2 THEN #silnikPredkoscPrzeliczona := #stacjaA_silnik_prędkość / 2.0; END_IF;
   IF NOT #setAwaria2 AND NOT #setAwaria3 THEN
       #silnikPredkoscPrzeliczona := #stacjaA_silnik_prędkość;
   END_IF;
END_REGION

REGION Network 6: Zablokowanie przejścia z trybu Manualne do Automatycznego
   RUNG wire#powerrail
      Contact( #resetAuto1 )
      wire#w1
      Coil( #blokadaPowrotuDoAuto )
   END_RUNG
   RUNG wire#powerrail
      Contact( #resetAuto2 )
   END_RUNG wire#w1
   // the same network as SCL:
   #blokadaPowrotuDoAuto := #resetAuto1 OR #resetAuto2;
END_REGION

REGION Network 7: Przełączenie na tryb Manualny
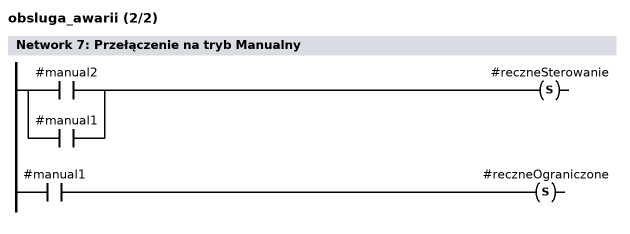
   RUNG wire#powerrail
      Contact( #manual2 )
      wire#w1
      S_Coil( #reczneSterowanie )
   END_RUNG
   RUNG wire#powerrail
      Contact( #manual1 )
   END_RUNG wire#w1
   RUNG wire#powerrail
      Contact( #manual1 )
      S_Coil( #reczneOgraniczone )
   END_RUNG
   // the same network as SCL:
   IF #manual2 OR #manual1 THEN #reczneSterowanie := TRUE; END_IF;
   IF #manual1 THEN #reczneOgraniczone := TRUE; END_IF;
END_REGION
END_FUNCTION_BLOCK

FUNCTION_BLOCK "obsluga_awarii_polinka"   // FB3, LAD
{ S7_Optimized_Access := 'TRUE' }
VERSION : 0.1
   VAR_TEMP   // added for the SCL form of the ladder/FBD networks
      _w1 : Bool;
   END_VAR
BEGIN

REGION Network 1
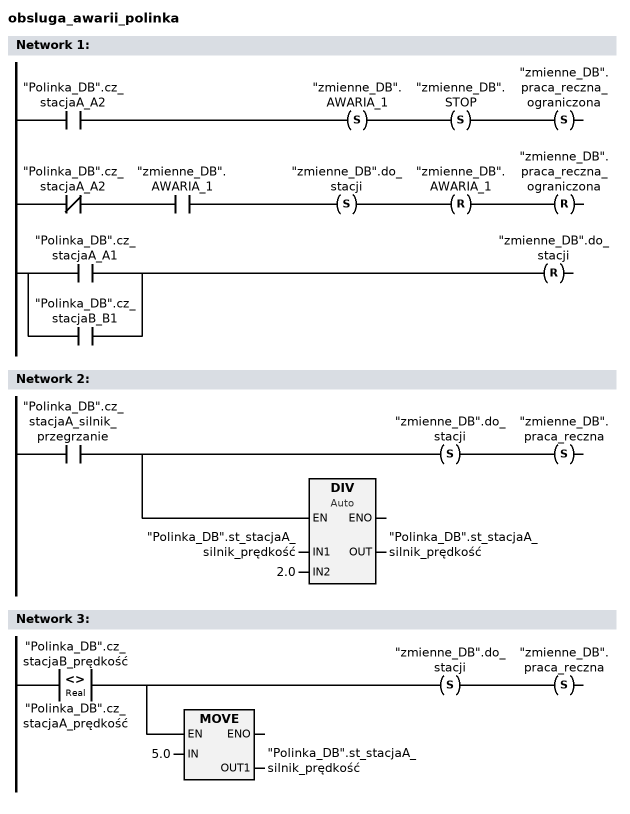
   RUNG wire#powerrail
      Contact( "Polinka_DB".cz_stacjaA_A2 )
      S_Coil( "zmienne_DB".AWARIA_1 )
      S_Coil( "zmienne_DB".STOP )
      S_Coil( "zmienne_DB".praca_reczna_ograniczona )
   END_RUNG
   RUNG wire#powerrail
      I_Contact( "Polinka_DB".cz_stacjaA_A2 )
      Contact( "zmienne_DB".AWARIA_1 )
      S_Coil( "zmienne_DB".do_stacji )
      R_Coil( "zmienne_DB".AWARIA_1 )
      R_Coil( "zmienne_DB".praca_reczna_ograniczona )
   END_RUNG
   RUNG wire#powerrail
      Contact( "Polinka_DB".cz_stacjaA_A1 )
      wire#w1
      R_Coil( "zmienne_DB".do_stacji )
   END_RUNG
   RUNG wire#powerrail
      Contact( "Polinka_DB".cz_stacjaB_B1 )
   END_RUNG wire#w1
   // the same network as SCL:
   IF "Polinka_DB".cz_stacjaA_A2 THEN
       "zmienne_DB".AWARIA_1 := TRUE;
       "zmienne_DB".STOP := TRUE;
       "zmienne_DB".praca_reczna_ograniczona := TRUE;
   END_IF;
   IF NOT "Polinka_DB".cz_stacjaA_A2 AND "zmienne_DB".AWARIA_1 THEN "zmienne_DB".do_stacji := TRUE; END_IF;
   #_w1 := NOT "Polinka_DB".cz_stacjaA_A2 AND "zmienne_DB".AWARIA_1;
   IF #_w1 THEN
       "zmienne_DB".AWARIA_1 := FALSE;
       "zmienne_DB".praca_reczna_ograniczona := FALSE;
   END_IF;
   IF "Polinka_DB".cz_stacjaA_A1 OR "Polinka_DB".cz_stacjaB_B1 THEN "zmienne_DB".do_stacji := FALSE; END_IF;
END_REGION

REGION Network 2
   RUNG wire#powerrail
      Contact( "Polinka_DB".cz_stacjaA_silnik_przegrzanie )
      wire#w1
      S_Coil( "zmienne_DB".do_stacji )
      S_Coil( "zmienne_DB".praca_reczna )
   END_RUNG
   RUNG wire#w1
      Div(in1 := "Polinka_DB".st_stacjaA_silnik_prędkość, in2 := 2.0, out => "Polinka_DB".st_stacjaA_silnik_prędkość)
   END_RUNG
   // the same network as SCL:
   IF "Polinka_DB".cz_stacjaA_silnik_przegrzanie THEN
       "zmienne_DB".do_stacji := TRUE;
       "zmienne_DB".praca_reczna := TRUE;
       "Polinka_DB".st_stacjaA_silnik_prędkość := "Polinka_DB".st_stacjaA_silnik_prędkość / 2.0;
   END_IF;
END_REGION

REGION Network 3
   RUNG wire#powerrail
      { S7_Templates := "SrcType := Real" } NE_Contact(in1 := "Polinka_DB".cz_stacjaB_prędkość, in2 := "Polinka_DB".cz_stacjaA_prędkość)
      wire#w1
      S_Coil( "zmienne_DB".do_stacji )
      S_Coil( "zmienne_DB".praca_reczna )
   END_RUNG
   RUNG wire#w1
      Move(in := 5.0, out1 => "Polinka_DB".st_stacjaA_silnik_prędkość)
   END_RUNG
   // the same network as SCL:
   IF "Polinka_DB".cz_stacjaB_prędkość <> "Polinka_DB".cz_stacjaA_prędkość THEN
       "zmienne_DB".do_stacji := TRUE;
       "zmienne_DB".praca_reczna := TRUE;
       "Polinka_DB".st_stacjaA_silnik_prędkość := 5.0;
   END_IF;
END_REGION

REGION Network 4 (SCL)
   IF "Polinka_DB".cz_stacjaA_prędkość*3.0 = "Polinka_DB"."cz_stacjaA_prędkość_(silnik)" AND "Polinka_DB".cz_stacjaA_prędkość <> 0 THEN
       "zmienne_DB".AWARIA_4 := 1;
       "zmienne_DB".STOP := 1;
       "zmienne_DB".praca_reczna_ograniczona := 1;
   ELSIF "zmienne_DB".AWARIA_4 = 1 THEN
       "zmienne_DB".AWARIA_4 := 0;
       "zmienne_DB".do_stacji := 1;
       "zmienne_DB".praca_reczna_ograniczona := 0;
   END_IF;
END_REGION
END_FUNCTION_BLOCK

FUNCTION "praca_reczna" : Void   // FC1, LAD
{ S7_Optimized_Access := 'TRUE' }
VERSION : 0.1
   VAR_TEMP   // added for the SCL form of the ladder/FBD networks
      _w1 : Bool;
      _w2 : Bool;
      _w3 : Bool;
      _w4 : Bool;
   END_VAR
BEGIN

REGION Network 1
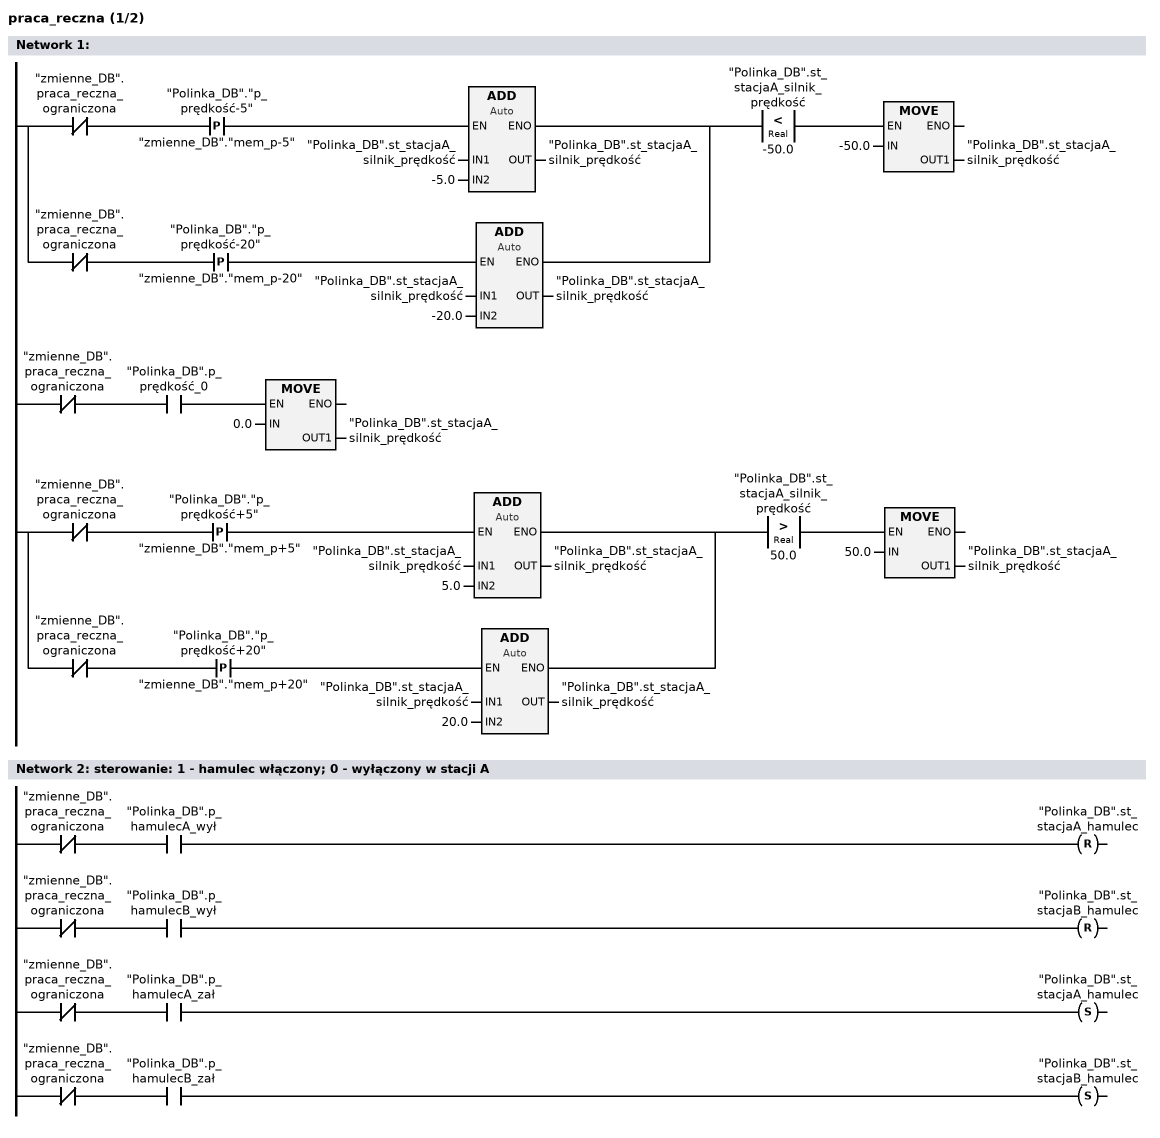
   RUNG wire#powerrail
      I_Contact( "zmienne_DB".praca_reczna_ograniczona )
      P_Contact(operand := "Polinka_DB"."p_prędkość-5", bit := "zmienne_DB"."mem_p-5")
      Add(in1 := "Polinka_DB".st_stacjaA_silnik_prędkość, in2 := -5.0, out => "Polinka_DB".st_stacjaA_silnik_prędkość)
      wire#w1
      { S7_Templates := "SrcType := Real" } LT_Contact(in1 := "Polinka_DB".st_stacjaA_silnik_prędkość, in2 := -50.0)
      Move(in := -50.0, out1 => "Polinka_DB".st_stacjaA_silnik_prędkość)
   END_RUNG
   RUNG wire#powerrail
      I_Contact( "zmienne_DB".praca_reczna_ograniczona )
      P_Contact(operand := "Polinka_DB"."p_prędkość-20", bit := "zmienne_DB"."mem_p-20")
      Add(in1 := "Polinka_DB".st_stacjaA_silnik_prędkość, in2 := -20.0, out => "Polinka_DB".st_stacjaA_silnik_prędkość)
   END_RUNG wire#w1
   RUNG wire#powerrail
      I_Contact( "zmienne_DB".praca_reczna_ograniczona )
      Contact( "Polinka_DB".p_prędkość_0 )
      Move(in := 0.0, out1 => "Polinka_DB".st_stacjaA_silnik_prędkość)
   END_RUNG
   RUNG wire#powerrail
      I_Contact( "zmienne_DB".praca_reczna_ograniczona )
      P_Contact(operand := "Polinka_DB"."p_prędkość+5", bit := "zmienne_DB"."mem_p+5")
      Add(in1 := "Polinka_DB".st_stacjaA_silnik_prędkość, in2 := 5.0, out => "Polinka_DB".st_stacjaA_silnik_prędkość)
      wire#w2
      { S7_Templates := "SrcType := Real" } GT_Contact(in1 := "Polinka_DB".st_stacjaA_silnik_prędkość, in2 := 50.0)
      Move(in := 50.0, out1 => "Polinka_DB".st_stacjaA_silnik_prędkość)
   END_RUNG
   RUNG wire#powerrail
      I_Contact( "zmienne_DB".praca_reczna_ograniczona )
      P_Contact(operand := "Polinka_DB"."p_prędkość+20", bit := "zmienne_DB"."mem_p+20")
      Add(in1 := "Polinka_DB".st_stacjaA_silnik_prędkość, in2 := 20.0, out => "Polinka_DB".st_stacjaA_silnik_prędkość)
   END_RUNG wire#w2
   // the same network as SCL:
   #_w1 := NOT "zmienne_DB".praca_reczna_ograniczona AND "Polinka_DB"."p_prędkość-5" AND NOT "zmienne_DB"."mem_p-5";   // rising edge of "Polinka_DB"."p_prędkość-5"
   "zmienne_DB"."mem_p-5" := "Polinka_DB"."p_prędkość-5";
   IF #_w1 THEN
       "Polinka_DB".st_stacjaA_silnik_prędkość := "Polinka_DB".st_stacjaA_silnik_prędkość + (-5.0);
   END_IF;
   #_w2 := NOT "zmienne_DB".praca_reczna_ograniczona AND "Polinka_DB"."p_prędkość-20" AND NOT "zmienne_DB"."mem_p-20";   // rising edge of "Polinka_DB"."p_prędkość-20"
   "zmienne_DB"."mem_p-20" := "Polinka_DB"."p_prędkość-20";
   IF #_w2 THEN
       "Polinka_DB".st_stacjaA_silnik_prędkość := "Polinka_DB".st_stacjaA_silnik_prędkość + (-20.0);
   END_IF;
   IF (#_w1 OR #_w2) AND ("Polinka_DB".st_stacjaA_silnik_prędkość < (-50.0)) THEN
       "Polinka_DB".st_stacjaA_silnik_prędkość := -50.0;
   END_IF;
   IF NOT "zmienne_DB".praca_reczna_ograniczona AND "Polinka_DB".p_prędkość_0 THEN
       "Polinka_DB".st_stacjaA_silnik_prędkość := 0.0;
   END_IF;
   #_w3 := NOT "zmienne_DB".praca_reczna_ograniczona AND "Polinka_DB"."p_prędkość+5" AND NOT "zmienne_DB"."mem_p+5";   // rising edge of "Polinka_DB"."p_prędkość+5"
   "zmienne_DB"."mem_p+5" := "Polinka_DB"."p_prędkość+5";
   IF #_w3 THEN
       "Polinka_DB".st_stacjaA_silnik_prędkość := "Polinka_DB".st_stacjaA_silnik_prędkość + 5.0;
   END_IF;
   #_w4 := NOT "zmienne_DB".praca_reczna_ograniczona AND "Polinka_DB"."p_prędkość+20" AND NOT "zmienne_DB"."mem_p+20";   // rising edge of "Polinka_DB"."p_prędkość+20"
   "zmienne_DB"."mem_p+20" := "Polinka_DB"."p_prędkość+20";
   IF #_w4 THEN
       "Polinka_DB".st_stacjaA_silnik_prędkość := "Polinka_DB".st_stacjaA_silnik_prędkość + 20.0;
   END_IF;
   IF (#_w3 OR #_w4) AND ("Polinka_DB".st_stacjaA_silnik_prędkość > 50.0) THEN
       "Polinka_DB".st_stacjaA_silnik_prędkość := 50.0;
   END_IF;
END_REGION

REGION Network 2: sterowanie: 1 - hamulec włączony; 0 - wyłączony w stacji A
   RUNG wire#powerrail
      I_Contact( "zmienne_DB".praca_reczna_ograniczona )
      Contact( "Polinka_DB".p_hamulecA_wył )
      R_Coil( "Polinka_DB".st_stacjaA_hamulec )
   END_RUNG
   RUNG wire#powerrail
      I_Contact( "zmienne_DB".praca_reczna_ograniczona )
      Contact( "Polinka_DB".p_hamulecB_wył )
      R_Coil( "Polinka_DB".st_stacjaB_hamulec )
   END_RUNG
   RUNG wire#powerrail
      I_Contact( "zmienne_DB".praca_reczna_ograniczona )
      Contact( "Polinka_DB".p_hamulecA_zał )
      S_Coil( "Polinka_DB".st_stacjaA_hamulec )
   END_RUNG
   RUNG wire#powerrail
      I_Contact( "zmienne_DB".praca_reczna_ograniczona )
      Contact( "Polinka_DB".p_hamulecB_zał )
      S_Coil( "Polinka_DB".st_stacjaB_hamulec )
   END_RUNG
   // the same network as SCL:
   IF NOT "zmienne_DB".praca_reczna_ograniczona AND "Polinka_DB".p_hamulecA_wył THEN
       "Polinka_DB".st_stacjaA_hamulec := FALSE;
   END_IF;
   IF NOT "zmienne_DB".praca_reczna_ograniczona AND "Polinka_DB".p_hamulecB_wył THEN
       "Polinka_DB".st_stacjaB_hamulec := FALSE;
   END_IF;
   IF NOT "zmienne_DB".praca_reczna_ograniczona AND "Polinka_DB".p_hamulecA_zał THEN
       "Polinka_DB".st_stacjaA_hamulec := TRUE;
   END_IF;
   IF NOT "zmienne_DB".praca_reczna_ograniczona AND "Polinka_DB".p_hamulecB_zał THEN
       "Polinka_DB".st_stacjaB_hamulec := TRUE;
   END_IF;
END_REGION

REGION Network 3: sterowanie: 1 - hamulec włączony; 0 - wyłączony w stacji A
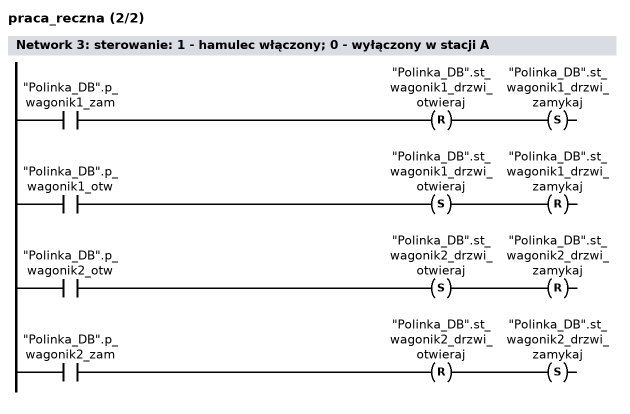
   RUNG wire#powerrail
      Contact( "Polinka_DB".p_wagonik1_zam )
      R_Coil( "Polinka_DB".st_wagonik1_drzwi_otwieraj )
      S_Coil( "Polinka_DB".st_wagonik1_drzwi_zamykaj )
   END_RUNG
   RUNG wire#powerrail
      Contact( "Polinka_DB".p_wagonik1_otw )
      S_Coil( "Polinka_DB".st_wagonik1_drzwi_otwieraj )
      R_Coil( "Polinka_DB".st_wagonik1_drzwi_zamykaj )
   END_RUNG
   RUNG wire#powerrail
      Contact( "Polinka_DB".p_wagonik2_otw )
      S_Coil( "Polinka_DB".st_wagonik2_drzwi_otwieraj )
      R_Coil( "Polinka_DB".st_wagonik2_drzwi_zamykaj )
   END_RUNG
   RUNG wire#powerrail
      Contact( "Polinka_DB".p_wagonik2_zam )
      R_Coil( "Polinka_DB".st_wagonik2_drzwi_otwieraj )
      S_Coil( "Polinka_DB".st_wagonik2_drzwi_zamykaj )
   END_RUNG
   // the same network as SCL:
   IF "Polinka_DB".p_wagonik1_zam THEN
       "Polinka_DB".st_wagonik1_drzwi_otwieraj := FALSE;
       "Polinka_DB".st_wagonik1_drzwi_zamykaj := TRUE;
   END_IF;
   IF "Polinka_DB".p_wagonik1_otw THEN
       "Polinka_DB".st_wagonik1_drzwi_otwieraj := TRUE;
       "Polinka_DB".st_wagonik1_drzwi_zamykaj := FALSE;
   END_IF;
   IF "Polinka_DB".p_wagonik2_otw THEN
       "Polinka_DB".st_wagonik2_drzwi_otwieraj := TRUE;
       "Polinka_DB".st_wagonik2_drzwi_zamykaj := FALSE;
   END_IF;
   IF "Polinka_DB".p_wagonik2_zam THEN
       "Polinka_DB".st_wagonik2_drzwi_otwieraj := FALSE;
       "Polinka_DB".st_wagonik2_drzwi_zamykaj := TRUE;
   END_IF;
END_REGION
END_FUNCTION

FUNCTION "sprawdzanie_pogody" : Void   // FC2, LAD
{ S7_Optimized_Access := 'TRUE' }
VERSION : 0.1
// Zadanie 3
   VAR_TEMP   // added for the SCL form of the ladder/FBD networks
      _w1 : Bool;
   END_VAR
BEGIN

REGION Network 1: Jeżeli bit ma stan wysoki to kolejka zostaje unieruchomiona na jedenj ze stacji
   // Popdunkt 2
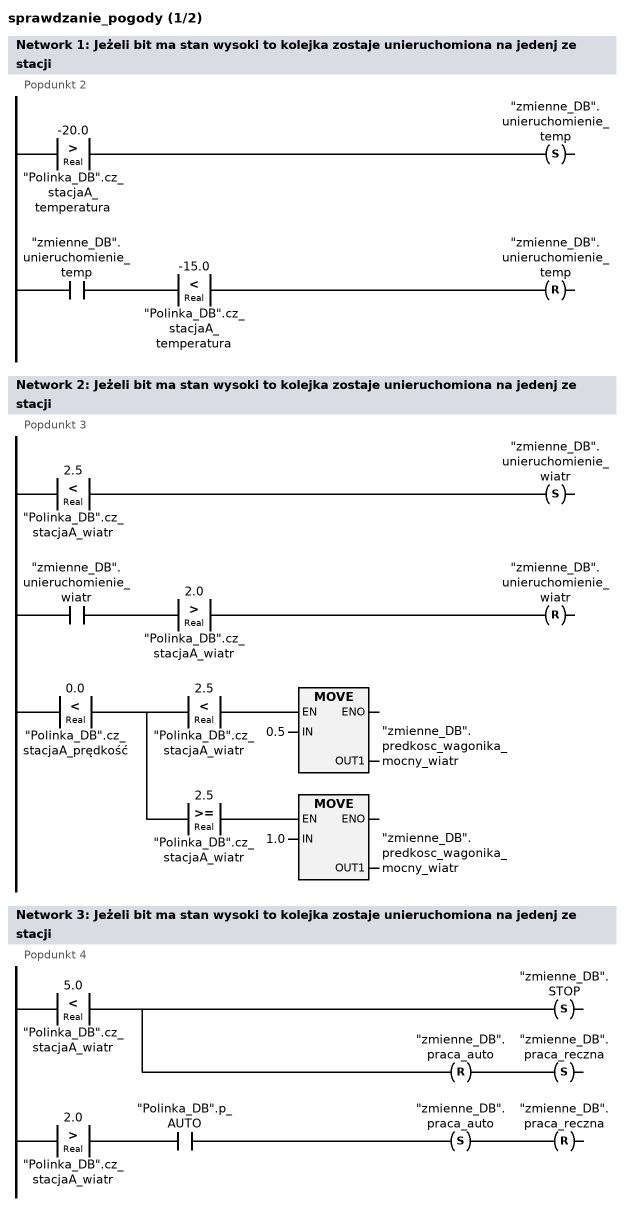
   RUNG wire#powerrail
      { S7_Templates := "SrcType := Real" } GT_Contact(in1 := -20.0, in2 := "Polinka_DB".cz_stacjaA_temperatura)
      S_Coil( "zmienne_DB".unieruchomienie_temp )
   END_RUNG
   RUNG wire#powerrail
      Contact( "zmienne_DB".unieruchomienie_temp )
      { S7_Templates := "SrcType := Real" } LT_Contact(in1 := -15.0, in2 := "Polinka_DB".cz_stacjaA_temperatura)
      R_Coil( "zmienne_DB".unieruchomienie_temp )
   END_RUNG
   // the same network as SCL:
   IF (-20.0) > "Polinka_DB".cz_stacjaA_temperatura THEN "zmienne_DB".unieruchomienie_temp := TRUE; END_IF;
   IF "zmienne_DB".unieruchomienie_temp AND ((-15.0) < "Polinka_DB".cz_stacjaA_temperatura) THEN
       "zmienne_DB".unieruchomienie_temp := FALSE;
   END_IF;
END_REGION

REGION Network 2: Jeżeli bit ma stan wysoki to kolejka zostaje unieruchomiona na jedenj ze stacji
   // Popdunkt 3
   RUNG wire#powerrail
      { S7_Templates := "SrcType := Real" } LT_Contact(in1 := 2.5, in2 := "Polinka_DB".cz_stacjaA_wiatr)
      S_Coil( "zmienne_DB".unieruchomienie_wiatr )
   END_RUNG
   RUNG wire#powerrail
      Contact( "zmienne_DB".unieruchomienie_wiatr )
      { S7_Templates := "SrcType := Real" } GT_Contact(in1 := 2.0, in2 := "Polinka_DB".cz_stacjaA_wiatr)
      R_Coil( "zmienne_DB".unieruchomienie_wiatr )
   END_RUNG
   RUNG wire#powerrail
      { S7_Templates := "SrcType := Real" } LT_Contact(in1 := 0.0, in2 := "Polinka_DB".cz_stacjaA_prędkość)
      wire#w1
      { S7_Templates := "SrcType := Real" } LT_Contact(in1 := 2.5, in2 := "Polinka_DB".cz_stacjaA_wiatr)
      Move(in := 0.5, out1 => "zmienne_DB".predkosc_wagonika_mocny_wiatr)
   END_RUNG
   RUNG wire#w1
      { S7_Templates := "SrcType := Real" } GE_Contact(in1 := 2.5, in2 := "Polinka_DB".cz_stacjaA_wiatr)
      Move(in := 1.0, out1 => "zmienne_DB".predkosc_wagonika_mocny_wiatr)
   END_RUNG
   // the same network as SCL:
   IF 2.5 < "Polinka_DB".cz_stacjaA_wiatr THEN "zmienne_DB".unieruchomienie_wiatr := TRUE; END_IF;
   IF "zmienne_DB".unieruchomienie_wiatr AND (2.0 > "Polinka_DB".cz_stacjaA_wiatr) THEN
       "zmienne_DB".unieruchomienie_wiatr := FALSE;
   END_IF;
   #_w1 := 0.0 < "Polinka_DB".cz_stacjaA_prędkość;
   IF #_w1 AND (2.5 < "Polinka_DB".cz_stacjaA_wiatr) THEN
       "zmienne_DB".predkosc_wagonika_mocny_wiatr := 0.5;
   END_IF;
   IF #_w1 AND (2.5 >= "Polinka_DB".cz_stacjaA_wiatr) THEN
       "zmienne_DB".predkosc_wagonika_mocny_wiatr := 1.0;
   END_IF;
END_REGION

REGION Network 3: Jeżeli bit ma stan wysoki to kolejka zostaje unieruchomiona na jedenj ze stacji
   // Popdunkt 4
   RUNG wire#powerrail
      { S7_Templates := "SrcType := Real" } LT_Contact(in1 := 5.0, in2 := "Polinka_DB".cz_stacjaA_wiatr)
      wire#w1
      S_Coil( "zmienne_DB".STOP )
   END_RUNG
   RUNG wire#w1
      R_Coil( "zmienne_DB".praca_auto )
      S_Coil( "zmienne_DB".praca_reczna )
   END_RUNG
   RUNG wire#powerrail
      { S7_Templates := "SrcType := Real" } GT_Contact(in1 := 2.0, in2 := "Polinka_DB".cz_stacjaA_wiatr)
      Contact( "Polinka_DB".p_AUTO )
      S_Coil( "zmienne_DB".praca_auto )
      R_Coil( "zmienne_DB".praca_reczna )
   END_RUNG
   // the same network as SCL:
   IF 5.0 < "Polinka_DB".cz_stacjaA_wiatr THEN
       "zmienne_DB".STOP := TRUE;
       "zmienne_DB".praca_auto := FALSE;
       "zmienne_DB".praca_reczna := TRUE;
   END_IF;
   IF (2.0 > "Polinka_DB".cz_stacjaA_wiatr) AND "Polinka_DB".p_AUTO THEN
       "zmienne_DB".praca_auto := TRUE;
       "zmienne_DB".praca_reczna := FALSE;
   END_IF;
END_REGION

REGION Network 4
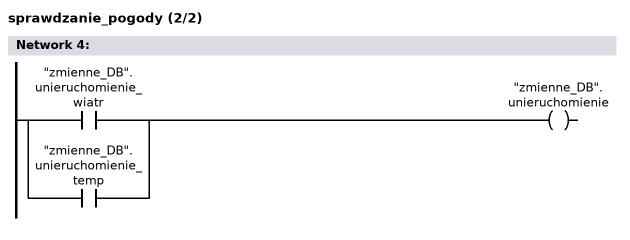
   RUNG wire#powerrail
      Contact( "zmienne_DB".unieruchomienie_wiatr )
      wire#w1
      Coil( "zmienne_DB".unieruchomienie )
   END_RUNG
   RUNG wire#powerrail
      Contact( "zmienne_DB".unieruchomienie_temp )
   END_RUNG wire#w1
   // the same network as SCL:
   "zmienne_DB".unieruchomienie := "zmienne_DB".unieruchomienie_wiatr OR "zmienne_DB".unieruchomienie_temp;
END_REGION
END_FUNCTION

ORGANIZATION_BLOCK "Main"   // OB1, LAD, ProgramCycle
TITLE = "Main Program Sweep (Cycle)"
{ S7_Optimized_Access := 'TRUE' }
VERSION : 0.1
   VAR_INPUT
      Initial_Call : Bool;   // Initial call of this OB
      Remanence : Bool;   // =True, if remanent data are available
   END_VAR
   VAR_TEMP   // added for the SCL form of the ladder/FBD networks
      _w1 : Bool;
      _w2 : Bool;
      _w3 : Bool;
   END_VAR
BEGIN

REGION Network 1: Pobieranie od modelu Polinka
   // Pobieraj tylko wtedy gdy nie masz odesłać danych oraz PUT został wykonany
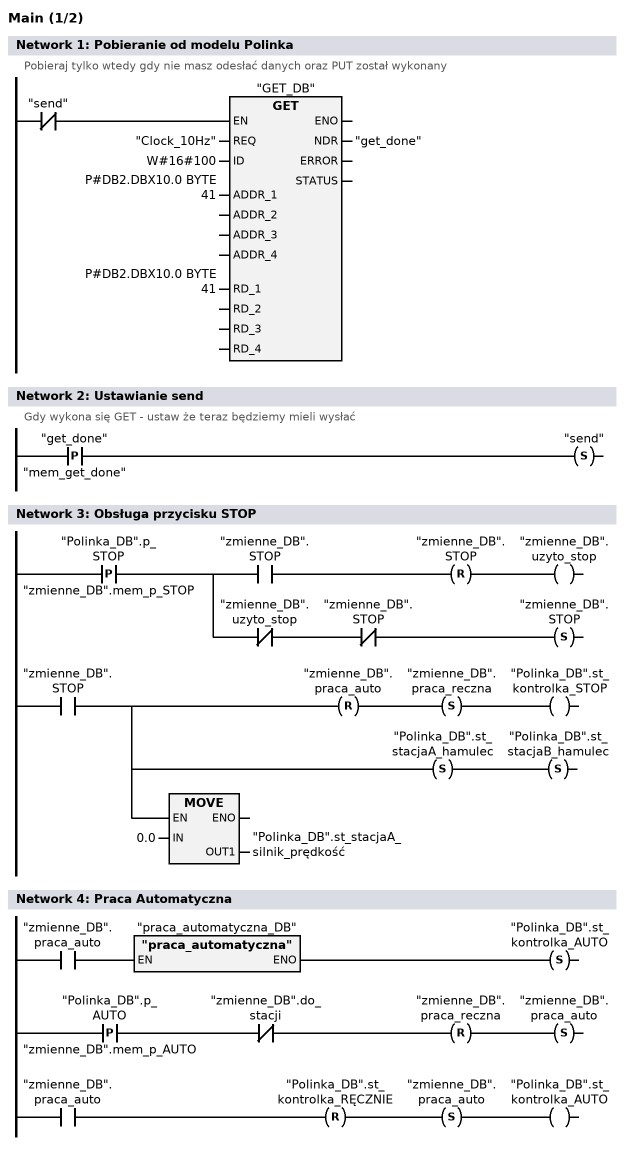
   IF NOT "send" THEN
       "GET_DB"(REQ := "Clock_10Hz",   // GET
                ID := W#16#100,
                ADDR_1 := P#DB2.DBX10.0 BYTE 41,
                RD_1 := P#DB2.DBX10.0 BYTE 41,
                NDR => "get_done");
   END_IF;
END_REGION

REGION Network 2: Ustawianie send
   // Gdy wykona się GET - ustaw że teraz będziemy mieli wysłać
   RUNG wire#powerrail
      P_Contact(operand := "get_done", bit := "mem_get_done")
      S_Coil( "send" )
   END_RUNG
   // the same network as SCL:
   #_w1 := "get_done" AND NOT "mem_get_done";   // rising edge of "get_done"
   "mem_get_done" := "get_done";
   IF #_w1 THEN "send" := TRUE; END_IF;
END_REGION

REGION Network 3: Obsługa przycisku STOP
   RUNG wire#powerrail
      P_Contact(operand := "Polinka_DB".p_STOP, bit := "zmienne_DB".mem_p_STOP)
      wire#w1
      Contact( "zmienne_DB".STOP )
      R_Coil( "zmienne_DB".STOP )
      Coil( "zmienne_DB".uzyto_stop )
   END_RUNG
   RUNG wire#w1
      I_Contact( "zmienne_DB".uzyto_stop )
      I_Contact( "zmienne_DB".STOP )
      S_Coil( "zmienne_DB".STOP )
   END_RUNG
   RUNG wire#powerrail
      Contact( "zmienne_DB".STOP )
      wire#w2
      R_Coil( "zmienne_DB".praca_auto )
      S_Coil( "zmienne_DB".praca_reczna )
      Coil( "Polinka_DB".st_kontrolka_STOP )
   END_RUNG
   RUNG wire#w2
      S_Coil( "Polinka_DB".st_stacjaA_hamulec )
      S_Coil( "Polinka_DB".st_stacjaB_hamulec )
   END_RUNG
   RUNG wire#w2
      Move(in := 0.0, out1 => "Polinka_DB".st_stacjaA_silnik_prędkość)
   END_RUNG
   // the same network as SCL:
   #_w1 := "Polinka_DB".p_STOP AND NOT "zmienne_DB".mem_p_STOP;   // rising edge of "Polinka_DB".p_STOP
   "zmienne_DB".mem_p_STOP := "Polinka_DB".p_STOP;
   #_w2 := #_w1 AND "zmienne_DB".STOP;
   IF #_w2 THEN "zmienne_DB".STOP := FALSE; END_IF;
   "zmienne_DB".uzyto_stop := #_w2;
   IF #_w1 AND NOT "zmienne_DB".uzyto_stop AND NOT "zmienne_DB".STOP THEN "zmienne_DB".STOP := TRUE; END_IF;
   IF "zmienne_DB".STOP THEN
       "zmienne_DB".praca_auto := FALSE;
       "zmienne_DB".praca_reczna := TRUE;
   END_IF;
   "Polinka_DB".st_kontrolka_STOP := "zmienne_DB".STOP;
   IF "zmienne_DB".STOP THEN
       "Polinka_DB".st_stacjaA_hamulec := TRUE;
       "Polinka_DB".st_stacjaB_hamulec := TRUE;
       "Polinka_DB".st_stacjaA_silnik_prędkość := 0.0;
   END_IF;
END_REGION

REGION Network 4: Praca Automatyczna
   RUNG wire#powerrail
      Contact( "zmienne_DB".praca_auto )
      "praca_automatyczna_DB"()
      S_Coil( "Polinka_DB".st_kontrolka_AUTO )
   END_RUNG
   RUNG wire#powerrail
      P_Contact(operand := "Polinka_DB".p_AUTO, bit := "zmienne_DB".mem_p_AUTO)
      I_Contact( "zmienne_DB".do_stacji )
      R_Coil( "zmienne_DB".praca_reczna )
      S_Coil( "zmienne_DB".praca_auto )
   END_RUNG
   RUNG wire#powerrail
      Contact( "zmienne_DB".praca_auto )
      R_Coil( "Polinka_DB".st_kontrolka_RĘCZNIE )
      S_Coil( "zmienne_DB".praca_auto )
      Coil( "Polinka_DB".st_kontrolka_AUTO )
   END_RUNG
   // the same network as SCL:
   "praca_automatyczna_DB"(EN := "zmienne_DB".praca_auto, ENO => #_w1);   // "praca_automatyczna"
   IF #_w1 THEN "Polinka_DB".st_kontrolka_AUTO := TRUE; END_IF;
   #_w2 := "Polinka_DB".p_AUTO AND NOT "zmienne_DB".mem_p_AUTO;   // rising edge of "Polinka_DB".p_AUTO
   "zmienne_DB".mem_p_AUTO := "Polinka_DB".p_AUTO;
   IF #_w2 AND NOT "zmienne_DB".do_stacji THEN
       "zmienne_DB".praca_reczna := FALSE;
       "zmienne_DB".praca_auto := TRUE;
   END_IF;
   IF "zmienne_DB".praca_auto THEN "Polinka_DB".st_kontrolka_RĘCZNIE := FALSE; END_IF;
   #_w3 := "zmienne_DB".praca_auto;
   IF #_w3 THEN "zmienne_DB".praca_auto := TRUE; END_IF;
   "Polinka_DB".st_kontrolka_AUTO := #_w3;
END_REGION

REGION Network 5: Praca Ręczna
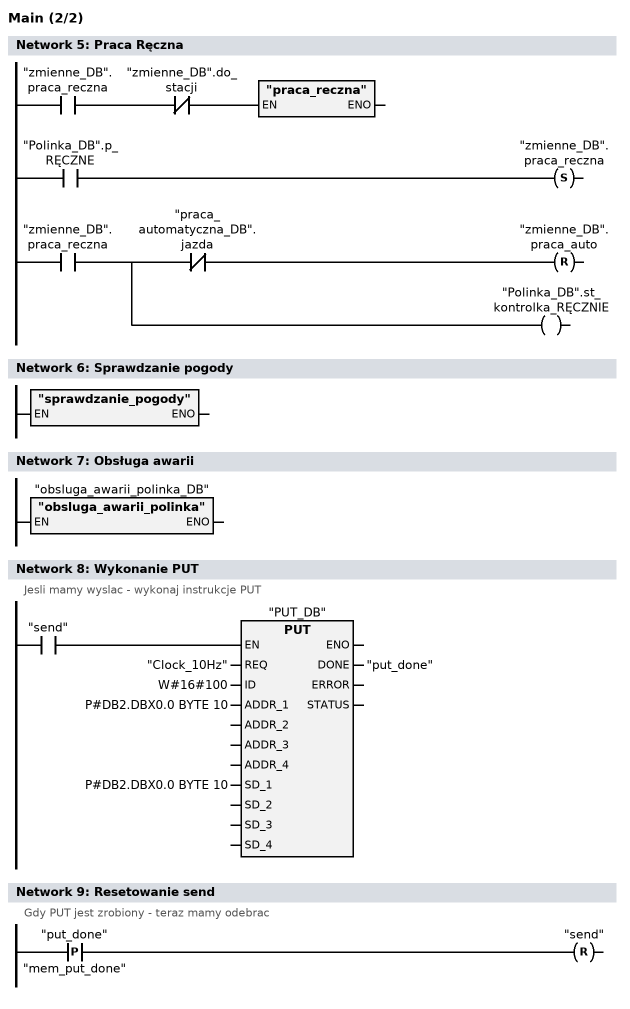
   RUNG wire#powerrail
      Contact( "zmienne_DB".praca_reczna )
      I_Contact( "zmienne_DB".do_stacji )
      "praca_reczna"()
   END_RUNG
   RUNG wire#powerrail
      Contact( "Polinka_DB".p_RĘCZNE )
      S_Coil( "zmienne_DB".praca_reczna )
   END_RUNG
   RUNG wire#powerrail
      Contact( "zmienne_DB".praca_reczna )
      wire#w1
      I_Contact( "praca_automatyczna_DB".jazda )
      R_Coil( "zmienne_DB".praca_auto )
   END_RUNG
   RUNG wire#w1
      Coil( "Polinka_DB".st_kontrolka_RĘCZNIE )
   END_RUNG
   // the same network as SCL:
   IF "zmienne_DB".praca_reczna AND NOT "zmienne_DB".do_stacji THEN "praca_reczna"(); END_IF;
   IF "Polinka_DB".p_RĘCZNE THEN "zmienne_DB".praca_reczna := TRUE; END_IF;
   IF "zmienne_DB".praca_reczna AND NOT "praca_automatyczna_DB".jazda THEN
       "zmienne_DB".praca_auto := FALSE;
   END_IF;
   "Polinka_DB".st_kontrolka_RĘCZNIE := "zmienne_DB".praca_reczna;
END_REGION

REGION Network 6: Sprawdzanie pogody
   RUNG wire#powerrail
      "sprawdzanie_pogody"()
   END_RUNG
   // the same network as SCL:
   "sprawdzanie_pogody"();
END_REGION

REGION Network 7: Obsługa awarii
   RUNG wire#powerrail
      "obsluga_awarii_polinka_DB"()
   END_RUNG
   // the same network as SCL:
   "obsluga_awarii_polinka_DB"();   // "obsluga_awarii_polinka"
END_REGION

REGION Network 8: Wykonanie PUT
   // Jesli mamy wyslac - wykonaj instrukcje PUT
   IF "send" THEN
       "PUT_DB"(REQ := "Clock_10Hz",   // PUT
                ID := W#16#100,
                ADDR_1 := P#DB2.DBX0.0 BYTE 10,
                SD_1 := P#DB2.DBX0.0 BYTE 10,
                DONE => "put_done");
   END_IF;
END_REGION

REGION Network 9: Resetowanie send
   // Gdy PUT jest zrobiony - teraz mamy odebrac
   RUNG wire#powerrail
      P_Contact(operand := "put_done", bit := "mem_put_done")
      R_Coil( "send" )
   END_RUNG
   // the same network as SCL:
   #_w1 := "put_done" AND NOT "mem_put_done";   // rising edge of "put_done"
   "mem_put_done" := "put_done";
   IF #_w1 THEN "send" := FALSE; END_IF;
END_REGION
END_ORGANIZATION_BLOCK

(* ===== HMI "HMI_RT_1" =====
system functions are stored by id; their names below are inferred from use
connection "HMI_Connection_1": ETHERNET, SMART_S7_1200_OMS

HMI tags "Default tag table"
   "DB_w1_x" : Int = PLC "DB".w1_x, 100 ms
   "DB_w1_y" : Int = PLC "DB".w1_y, 100 ms
   "DB_w1_drzwiP_dx" : Int = PLC "DB".w1_drzwiP_dx, 100 ms
   "DB_zero" : Int = PLC "DB".zero, 100 ms
   "DB_w1_drzwiL_dx" : Int = PLC "DB".w1_drzwiL_dx, 100 ms
   "DB_w1_liczba_pasażerów" : Int = PLC "DB".w1_liczba_pasażerów, 100 ms
   "DB_w2_x" : Int = PLC "DB".w2_x, 100 ms
   "DB_w2_y" : Int = PLC "DB".w2_y, 100 ms
   "DB_w2_drzwiP_dx" : Int = PLC "DB".w2_drzwiP_dx, 100 ms
   "DB_w2_drzwiL_dx" : Int = PLC "DB".w2_drzwiL_dx, 100 ms
   "DB_w2_liczba_pasażerów" : Int = PLC "DB".w2_liczba_pasażerów, 100 ms
   "DB_prędkość_wiatru" : Real = PLC "DB".prędkość_wiatru, 100 ms
   "DB_temperatura" : Real = PLC "DB".temperatura, 100 ms
   "DB_w1_drzwi_zamknięte" : Bool = PLC "DB".w1_drzwi_zamknięte, 100 ms
   "DB_czas_do_odjazdu" : Int = PLC "DB".czas_do_odjazdu, 100 ms
   "DB_stacjaA_silnik_prędkość_odczytana" : Real = PLC "DB".stacjaA_silnik_prędkość_odczytana, 100 ms
   "DB_stacjaA_cz_A1" : Bool = PLC "DB".stacjaA_cz_A1, 100 ms
   "DB_stacjaA_cz_A2" : Bool = PLC "DB".stacjaA_cz_A2, 100 ms
   "DB_stacjaB_cz_B2" : Bool = PLC "DB".stacjaB_cz_B2, 100 ms
   "DB_stacjaB_cz_B1" : Bool = PLC "DB".stacjaB_cz_B1, 100 ms
   "DB_stacjaA_hamulec" : Bool = PLC "DB".stacjaA_hamulec, 100 ms
   "DB_stacjaB_hamulec" : Bool = PLC "DB".stacjaB_hamulec, 100 ms
   "Polinka_DB_st_stacjaA_czerwone" : Bool = PLC Polinka_DB.st_stacjaA_czerwone AT %DB2.DBX4.2, 100 ms
   "Polinka_DB_st_stacjaA_zielone" : Bool = PLC Polinka_DB.st_stacjaA_zielone AT %DB2.DBX4.1, 100 ms
   "DB_stacjaA_pasażer_0" : Bool = PLC "DB".stacjaA_pasażer_0, 100 ms
   "DB_stacjaA_pasażer-1" : Bool = PLC "DB".stacjaA_pasażer-1, 100 ms
   "DB_stacjaA_pasażer+1" : Bool = PLC "DB".stacjaA_pasażer+1, 100 ms
   "DB_stacjaA_pasażerDOWN" : Bool = PLC "DB".stacjaA_pasażerDOWN, 100 ms
   "DB_stacjaA_pasażerUP" : Bool = PLC "DB".stacjaA_pasażerUP, 100 ms
   "Polinka_DB_st_stacjaB_czerwone" : Bool = PLC Polinka_DB.st_stacjaB_czerwone AT %DB2.DBX4.5, 100 ms
   "Polinka_DB_st_stacjaB_zielone" : Bool = PLC Polinka_DB.st_stacjaB_zielone AT %DB2.DBX4.4, 100 ms
   "DB_stacjaB_pasażer+1" : Bool = PLC "DB".stacjaB_pasażer+1, 500 ms
   "DB_stacjaB_pasażer-1" : Bool = PLC "DB".stacjaB_pasażer-1, 500 ms
   "DB_stacjaB_pasażer_0" : Bool = PLC "DB".stacjaB_pasażer_0, 500 ms
   "DB_stacjaB_pasażerDOWN" : Bool = PLC "DB".stacjaB_pasażerDOWN, 100 ms
   "DB_stacjaB_pasażerUP" : Bool = PLC "DB".stacjaB_pasażerUP, 100 ms
   "Polinka_DB_p_prędkość-20" : Bool = PLC Polinka_DB.p_prędkość-20 AT %DB2.DBX48.5, 100 ms
   "DB_klawiatura" : Word = PLC "DB".klawiatura, 100 ms
   "Polinka_DB_cz_wagonik1_położenie" : Real = PLC Polinka_DB.cz_wagonik1_położenie AT %DB2.DBD10, 100 ms
   "DB_w1_d" : Real = PLC "DB".w1_d, 100 ms
   "Polinka_DB_cz_wagonik1_DZ" : Bool = PLC Polinka_DB.cz_wagonik1_DZ AT %DB2.DBX16.0, 100 ms
   "Polinka_DB_cz_wagonik1_DO" : Bool = PLC Polinka_DB.cz_wagonik1_DO AT %DB2.DBX16.1, 100 ms
   "DB_w2_d" : Real = PLC "DB".w2_d, 100 ms
   "Polinka_DB_cz_wagonik2_DZ" : Bool = PLC Polinka_DB.cz_wagonik2_DZ AT %DB2.DBX24.0, 100 ms
   "Polinka_DB_cz_wagonik2_DO" : Bool = PLC Polinka_DB.cz_wagonik2_DO AT %DB2.DBX24.1, 100 ms
   "Polinka_DB_cz_stacjaA_silnik_przegrzanie" : Bool = PLC Polinka_DB.cz_stacjaA_silnik_przegrzanie AT %DB2.DBX42.0, 100 ms
   "Polinka_DB_st_stacjaA_hamulec" : Bool = PLC Polinka_DB.st_stacjaA_hamulec AT %DB2.DBX4.0, 100 ms
   "Polinka_DB_cz_stacjaA_prędkość" : Real = PLC Polinka_DB.cz_stacjaA_prędkość AT %DB2.DBD30, 100 ms
   "Polinka_DB_cz_stacjaA_prędkość_(silnik)" : Real = PLC Polinka_DB.cz_stacjaA_prędkość_(silnik) AT %DB2.DBD26, 100 ms
   "DB_stacjaA_prędkość_odczytana" : Real = PLC "DB".stacjaA_prędkość_odczytana, 100 ms
   "DB_stacjaB_prędkość_odczytana" : Real = PLC "DB".stacjaB_prędkość_odczytana, 100 ms
   "DB_awaria1" : Bool = PLC "DB".awaria1, 100 ms
   "DB_awaria2" : Bool = PLC "DB".awaria2, 100 ms
   "DB_awaria5" : Bool = PLC "DB".awaria5, 100 ms
   "DB_awaria4" : Bool = PLC "DB".awaria4, 100 ms
   "DB_awaria3" : Bool = PLC "DB".awaria3, 100 ms
   "Polinka_DB_st_kontrolka_STOP" : Bool = PLC Polinka_DB.st_kontrolka_STOP AT %DB2.DBX8.0, 100 ms
   "Polinka_DB_st_kontrolka_AUTO" : Bool = PLC Polinka_DB.st_kontrolka_AUTO AT %DB2.DBX8.1, 100 ms
   "Polinka_DB_st_kontrolka_RĘCZNIE" : Bool = PLC Polinka_DB.st_kontrolka_RĘCZNIE AT %DB2.DBX8.2, 100 ms

screen "Polinka_Root" 800x480, template "Template_1"
   GraphicView "Graphic view_2" at 17,136 size 77x109; Picture "polinka_2_yellow_bez_drzwi_1"
      DirectMovement <- "DB_w1_x"
      DirectMovement <- "DB_w1_y"
   GraphicView "Graphic view_1" at 42,185 size 15x54; Picture "Polinka_drzwi_L"
      DirectMovement <- "DB_w1_drzwiL_dx"
      DirectMovement <- "DB_w1_y"
   GraphicView "Graphic view_3" at 55,185 size 15x54; Picture "Polinka_drzwi_P"
      DirectMovement <- "DB_w1_drzwiP_dx"
      DirectMovement <- "DB_w1_y"
   IOField "I/O field_1" at 41,183 size 30x37; FormatPattern 9
      DirectMovement <- "DB_w1_x"
      DirectMovement <- "DB_w1_y"
      ProcessValue <- "DB_w1_liczba_pasażerów"
   GraphicView "Graphic view_4" at 705,136 size 77x109; Picture "polinka_1_red_bez_drzwi"
      DirectMovement <- "DB_w2_x"
      DirectMovement <- "DB_w2_y"
   GraphicView "Graphic view_5" at 730,185 size 15x54; Picture "Polinka_drzwi_L"
      DirectMovement <- "DB_w2_drzwiL_dx"
      DirectMovement <- "DB_w2_y"
   GraphicView "Graphic view_6" at 743,185 size 15x54; Picture "Polinka_drzwi_P"
      DirectMovement <- "DB_w2_drzwiP_dx"
      DirectMovement <- "DB_w2_y"
   IOField "I/O field_2" at 729,183 size 30x37; FormatPattern 9
      DirectMovement <- "DB_w2_x"
      DirectMovement <- "DB_w2_y"
      ProcessValue <- "DB_w2_liczba_pasażerów"
   TextField "Text field_5" at 350,236 size 95x23; Text 'rzeka Odra'
   TextField "Text field_8" at 228,181 size 146x18; Text 'Prędkość wiatru [m/s]:'
   Button "Button_1" at 444,178 size 51x24; TextOff '-1 m/s'
      on Release: function_b9b71300("DB_prędkość_wiatru", 1)
   Button "Button_2" at 499,178 size 51x24; TextOff '+1 m/s'
      on Release: function_dd21b452("DB_prędkość_wiatru", 1)
   IOField "I/O field_3" at 374,180 size 64x21; FormatPattern 999.9
      ProcessValue <- "DB_prędkość_wiatru"
   TextField "Text field_9" at 228,209 size 149x18; Text 'Temp. powietrza [st.C]:'
   Button "Button_3" at 444,206 size 51x24; TextOff '-1 st.C'
      on Release: function_b9b71300("DB_temperatura", 1)
   Button "Button_4" at 499,206 size 51x24; TextOff '+1 st.C'
      on Release: function_dd21b452("DB_temperatura", 1)
   IOField "I/O field_4" at 388,207 size 50x21; FormatPattern 999.9
      ProcessValue <- "DB_temperatura"
   TextField "Text field_22" at 319,70 size 56x52; Text '3P'
   TextField "Text field_23" at 377,74 size 101x46; Text 'Programowanie Przemysłu Przyszłości'
   TextField "Text field_31" at 5,409 size 93x30; Text 'Pozycja wagonika1 [m]:'
   IOField "I/O field_7" at 99,422 size 49x16; FormatPattern s999.9
      ProcessValue <- "DB_w1_d"
   TextField "Text field_32" at 5,438 size 103x17; Text 'cz_wagonik1_DZ:'
   IOField "I/O field_8" at 111,440 size 19x16; FormatPattern 1
      ProcessValue <- "Polinka_DB_cz_wagonik1_DZ"
   TextField "Text field_33" at 5,456 size 104x17; Text 'cz_wagonik1_DO:'
   IOField "I/O field_9" at 111,458 size 19x16; FormatPattern 1
      ProcessValue <- "Polinka_DB_cz_wagonik1_DO"
   TextField "Text field_34" at 650,409 size 93x30; Text 'Pozycja wagonika2 [m]:'
   IOField "I/O field_10" at 746,422 size 46x16; FormatPattern s999.9
      ProcessValue <- "DB_w2_d"
   TextField "Text field_35" at 650,438 size 103x17; Text 'cz_wagonik2_DZ:'
   IOField "I/O field_11" at 757,440 size 19x16; FormatPattern 1
      ProcessValue <- "Polinka_DB_cz_wagonik2_DZ"
   TextField "Text field_36" at 650,456 size 104x17; Text 'cz_wagonik2_DO:'
   IOField "I/O field_12" at 757,458 size 19x16; FormatPattern 1
      ProcessValue <- "Polinka_DB_cz_wagonik2_DO"
   Group "Group_4" at 309,70 size 180x55
   Group "Group_1" at 705,136 size 77x109; Picture "polinka_1_red_bez_drzwi"
   TextField "Text field_3" at 9,0 size 78x24; Text 'Stacja A'
   TextField "Text field_4" at 718,0 size 72x24; Text 'Stacja B'
   TextField "Text field_6" at 715,19 size 84x17; Text 'Kampus Główny'
   TextField "Text field_7" at 1,19 size 96x17; Text 'Kampus "Na Grobli"'
   Group "Group_2" at 233,236 size 326x27
   Group "Group_3" at 228,178 size 322x52
   TextField "Text field_10" at 38,106 size 39x17; Text 'cz_A1'
      Appearance <- "DB_stacjaA_cz_A1"
   TextField "Text field_11" at 262,1 size 224x27; Text 'Czas do odjazdu [sek]:'
   IOField "I/O field_5" at 488,4 size 51x26; FormatPattern 999
      ProcessValue <- "DB_czas_do_odjazdu"
   TextField "Text field_12" at 573,6 size 38x17; Text 'cz_B2'
      Appearance <- "DB_stacjaB_cz_B2"
   TextField "Text field_13" at 188,7 size 39x17; Text 'cz_A2'
      Appearance <- "DB_stacjaA_cz_A2"
   TextField "Text field_14" at 726,104 size 38x17; Text 'cz_B1'
      Appearance <- "DB_stacjaB_cz_B1"
   Group "Group" at 17,136 size 77x109; Picture "polinka_2_yellow_bez_drzwi_1"
   Button "Button_5" at 65,321 size 45x24; TextOff '+1'
      on Release: SetBit("DB_stacjaA_pasażer+1")
   Circle "Circle_1" at 87,271 size 22x22
      Appearance <- "Polinka_DB_st_stacjaA_czerwone"
   Circle "Circle_2" at 87,296 size 22x22
      Appearance <- "Polinka_DB_st_stacjaA_zielone"
   Line "Line_15" at 74,273 size 0x41
      Appearance <- "DB_stacjaA_pasażerUP"
   Button "Button_9" at 9,321 size 45x24; TextOff '-1'
      on Release: SetBit("DB_stacjaA_pasażer-1")
   Line "Line_16" at 17,273 size 0x41
      Appearance <- "DB_stacjaA_pasażerDOWN"
   Button "Button_6" at 28,272 size 26x44; TextOff '0'
      on Release: SetBit("DB_stacjaA_pasażer_0")
   TextField "Text field_16" at 64,246 size 49x17; Text 'Wejście'
   TextField "Text field_17" at 9,246 size 49x17; Text 'Wyjście'
   Button "Button_7" at 691,321 size 45x24; TextOff '+1'
      on Release: SetBit("DB_stacjaB_pasażer+1")
   Circle "Circle_3" at 713,271 size 22x22
      Appearance <- "Polinka_DB_st_stacjaB_czerwone"
   Circle "Circle_4" at 713,296 size 22x22
      Appearance <- "Polinka_DB_st_stacjaB_zielone"
   Line "Line_17" at 700,273 size 0x41
      Appearance <- "DB_stacjaB_pasażerUP"
   Button "Button_8" at 747,321 size 45x24; TextOff '-1'
      on Release: SetBit("DB_stacjaB_pasażer-1")
   Line "Line_18" at 755,273 size 0x41
      Appearance <- "DB_stacjaB_pasażerDOWN"
   Button "Button_10" at 766,272 size 26x44; TextOff '0'
      on Release: SetBit("DB_stacjaB_pasażer_0")
   TextField "Text field_18" at 690,245 size 49x17; Text 'Wejście'
   TextField "Text field_19" at 747,245 size 49x17; Text 'Wyjście'
   TextField "Text field_20" at 17,350 size 80x18; Text 'Pasażerowie'
   TextField "Text field_21" at 700,349 size 80x18; Text 'Pasażerowie'
   Group "Group_7" at 650,409 size 146x67
   Group "Group_8" at 5,409 size 146x67
   TextField "Text field_2" at 6,42 size 74x17; Text 'Silnik [m/s]:'
   TextField "Text field_1" at 6,58 size 68x17; Text 'Hamulec A:'
   IOField "I/O field_6" at 80,44 size 45x14; FormatPattern s99.9
      ProcessValue <- "DB_stacjaA_silnik_prędkość_odczytana"
   SymbolicIOField "Symbolic I/O field_1" at 80,60 size 45x14; TextOff 'WYŁ'; TextOn 'ZAŁ'
      ProcessValue <- "DB_stacjaA_hamulec"
      Appearance <- "DB_stacjaA_hamulec"
   TextField "Text field_38" at 6,74 size 74x17; Text 'KołoA[m/s]:'
   IOField "I/O field_13" at 80,76 size 45x14; FormatPattern s99.9
      ProcessValue <- "DB_stacjaA_prędkość_odczytana"
   SymbolicIOField "Symbolic I/O field_3" at 131,45 size 30x13; TextOn 'ZAB'; TextOff '-'
      ProcessValue <- "Polinka_DB_cz_stacjaA_silnik_przegrzanie"
      Appearance <- "Polinka_DB_cz_stacjaA_silnik_przegrzanie"
   TextField "Text field_40" at 675,56 size 67x17; Text 'Hamulec B:'
   SymbolicIOField "Symbolic I/O field_4" at 749,58 size 45x14; TextOn 'ZAŁ'; TextOff 'WYŁ'
      ProcessValue <- "DB_stacjaB_hamulec"
      Appearance <- "DB_stacjaB_hamulec"
   TextField "Text field_41" at 675,72 size 73x17; Text 'KołoB[m/s]:'
   IOField "I/O field_15" at 749,74 size 45x14; FormatPattern s99.9
      ProcessValue <- "DB_stacjaB_prędkość_odczytana"
   Button "Button_21" at 540,320 size 73x24; TextOff 'Awaria_1'
      on Release: InvertBit("DB_awaria1")
      Appearance <- "DB_awaria1"
   TextField "Text field_37" at 518,275 size 108x19; Text 'Symulator awarii'
   Button "Button_26" at 541,350 size 73x24; TextOff 'Awaria_2'
      on Release: InvertBit("DB_awaria2")
      Appearance <- "DB_awaria2"
   Button "Button_29" at 541,379 size 73x24; TextOff 'Awaria_3'
      on Release: InvertBit("DB_awaria3")
      Appearance <- "DB_awaria3"
   Button "Button_30" at 541,409 size 73x24; TextOff 'Awaria_4'
      on Release: InvertBit("DB_awaria4")
      Appearance <- "DB_awaria4"
   Button "Button_31" at 541,439 size 73x24; TextOff 'Awaria_5'
      on Release: InvertBit("DB_awaria5")
      Appearance <- "DB_awaria5"
   Button "Button_11" at 249,320 size 45x24; TextOff '-20'
      on Press: function_b14e0dd5("DB_klawiatura", 3)
   Button "Button_13" at 183,361 size 56x29; TextOff 'AUTO'
      on Press: function_b14e0dd5("DB_klawiatura", 1)
      Appearance <- "Polinka_DB_st_kontrolka_AUTO"
   Button "Button_14" at 183,303 size 56x53; TextOff 'STOP'
      on Press: function_b14e0dd5("DB_klawiatura", 0)
      Appearance <- "Polinka_DB_st_kontrolka_STOP"
   Button "Button_15" at 183,410 size 56x29; TextOff 'RĘCZNIE'
      on Press: function_b14e0dd5("DB_klawiatura", 2)
      Appearance <- "Polinka_DB_st_kontrolka_RĘCZNIE"
   Button "Button_12" at 300,320 size 45x24; TextOff '-5'
      on Press: function_b14e0dd5("DB_klawiatura", 4)
   Button "Button_16" at 350,320 size 45x24; TextOff '0'
      on Press: function_b14e0dd5("DB_klawiatura", 5)
   Button "Button_17" at 399,320 size 45x24; TextOff '+5'
      on Press: function_b14e0dd5("DB_klawiatura", 6)
   Button "Button_18" at 449,320 size 45x24; TextOff '+20'
      on Press: function_b14e0dd5("DB_klawiatura", 7)
   TextField "Text field_24" at 264,301 size 201x18; Text 'Zadajnik prędkości silnika [m/s]:'
   Button "Button_19" at 250,376 size 45x24; TextOff 'ZAŁ'
      on Press: function_b14e0dd5("DB_klawiatura", 8)
   Button "Button_20" at 301,376 size 45x24; TextOff 'WYŁ'
      on Press: function_b14e0dd5("DB_klawiatura", 9)
   Button "Button_22" at 400,376 size 45x24; TextOff 'ZAŁ'
      on Press: function_b14e0dd5("DB_klawiatura", 10)
   Button "Button_23" at 450,376 size 45x24; TextOff 'WYŁ'
      on Press: function_b14e0dd5("DB_klawiatura", 11)
   TextField "Text field_25" at 265,357 size 73x18; Text 'Hamulec A:'
   Button "Button_24" at 249,446 size 45x24; TextOff 'OTW'
      on Press: function_b14e0dd5("DB_klawiatura", 12)
   Button "Button_25" at 300,446 size 45x24; TextOff 'ZAM'
      on Press: function_b14e0dd5("DB_klawiatura", 13)
   Button "Button_27" at 399,446 size 45x24; TextOff 'OTW'
      on Press: function_b14e0dd5("DB_klawiatura", 14)
   Button "Button_28" at 449,446 size 45x24; TextOff 'ZAM'
      on Press: function_b14e0dd5("DB_klawiatura", 15)
   TextField "Text field_26" at 308,412 size 137x18; Text 'Sterowanie drzwiami:'
   TextField "Text field_27" at 410,358 size 72x18; Text 'Hamulec B:'
   TextField "Text field_28" at 264,426 size 69x18; Text 'wagonik 1'
   TextField "Text field_29" at 412,427 size 69x18; Text 'wagonik 2'
   TextField "Text field_30" at 241,275 size 178x19; Text 'Panel operatorski w Stacji A'
*)